(* IEC 61131-3 sources: Yaha/Documentation/Infomaterial/OSCAT/pcworx_basic_333/module_export (part 4) *)

(* ---- FT_PIDW.ST ---- *)
(*@PROPERTIES_EX@
TYPE: POU
LOCALE: 0
IEC_LANGUAGE: ST
PLC_TYPE: independent
PROC_TYPE: independent
GROUP: ENGINEERING.CONTROL
*)
(*@KEY@:DESCRIPTION*)
version 1.2	11. mar. 2009
programmer 	hugo
tested by	oscat

FT_PIDW is a PID controller with dynamic wind_up reset.
The PID controller works according to the fomula Y = KP *(IN + KI * INTEG(e) + DERIV(e) ).
a rst will reset the integrator to 0
lim_h and Lim_l set the possible output range of the internal integrator.
the output flags lim will signal that the output limits are active.

default values for KP = 1, KI = 1, ILIM_L = -1E37, iLIM_H = +1E38.
(*@KEY@:END_DESCRIPTION*)
FUNCTION_BLOCK FT_PIDW

(*Group:Default*)

VAR_INPUT
	IN :	REAL;
	KP :	REAL := 1.0;
	TN :	REAL := 1.0;
	TV :	REAL := 1.0;
	LIM_L :	REAL := -1.0E38;
	LIM_H :	REAL := 1.0E38;
	RST :	BOOL := FALSE;
END_VAR

VAR_OUTPUT
	Y :	REAL;
	LIM :	BOOL;
END_VAR

VAR
	integ :	INTEGRATE;
	diff :	FT_DERIV;
	YI :	REAL;
END_VAR

(*@KEY@: WORKSHEET
NAME: FT_PIDW
IEC_LANGUAGE: ST
*)
(* run the integrator *)
IF tn = 0.0 OR rst THEN
	integ(E := FALSE, Y := YI);
	YI := integ.Y;
	YI := 0.0;
ELSE
	integ(X := IN, K := 1.0 / TN, E := NOT LIM, Y := YI);
	YI := integ.Y;
END_IF;

(* add up integrator and linear part *)
Y := KP * (IN + YI);

(* run differentiator *)
diff(IN := IN, K := TV);

(* set lim before differentiator is added to stop integrator if necessary *)
IF Y > LIM_L AND Y < LIM_H THEN
	LIM := FALSE;
ELSE
	LIM := TRUE;
END_IF;

(* add differential part and limit output Y *)

Y := LIMIT(LIM_L, Y + KP * diff.out, LIM_H);

(* revision history
hm 3. jun. 2008 	rev 1.0
	original version

hm	5. nov. 2008	rev 1.1
	changed code to use integrate

hm	11. mar. 2009	rev 1.2
	real constants updated to new systax using dot

*)
(*@KEY@: END_WORKSHEET *)
END_FUNCTION_BLOCK

(* ---- FT_PIDWL.ST ---- *)
(*@PROPERTIES_EX@
TYPE: POU
LOCALE: 0
IEC_LANGUAGE: ST
PLC_TYPE: independent
PROC_TYPE: independent
GROUP: ENGINEERING.CONTROL
*)
(*@KEY@:DESCRIPTION*)
version 1.3	13. nov. 2009
programmer 	hugo
tested by	tobias

FT_PIDWL is a PID controller with dynamic wind_up reset.
The PID controller works according to the fomula Y = KP *(IN + KI * INTEG(e) + DERIV(e) ).
a rst will reset the integrator to 0
lim_h and Lim_l set the possible output range of the internal integrator.
the output flags lim will signal that the output limits are active.

default values for KP = 1, KI = 1, ILIM_L = -1E37, iLIM_H = +1E38.
(*@KEY@:END_DESCRIPTION*)
FUNCTION_BLOCK FT_PIDWL

(*Group:Default*)

VAR_INPUT
	IN :	REAL;
	KP :	REAL := 1.0;
	TN :	REAL := 1.0;
	TV :	REAL := 1.0;
	LIM_L :	REAL := -1.0E38;
	LIM_H :	REAL := 1.0E38;
	RST :	BOOL;
END_VAR

VAR_OUTPUT
	Y :	REAL;
	LIM :	BOOL;
END_VAR

VAR
	piwl :	FT_PIWL;
	diff :	FT_DERIV;
END_VAR

(*@KEY@: WORKSHEET
NAME: FT_PIDWL
IEC_LANGUAGE: ST
*)
(* if rst then *)
IF rst THEN
	piwl(rst := TRUE);
	piwl.RST := FALSE;
ELSE
	(* run PIWL controller first *)
	(* we need to check if TN = 0 and do alternative calls *)
	IF TN = 0.0 THEN
		piwl(in := IN * KP, KP := 1.0, KI := 0.0, LIM_L := LIM_L, LIM_H := LIM_H);
	ELSE
		piwl(in := IN * KP, KP := 1.0, KI := 1.0 / TN, LIM_L := LIM_L, LIM_H := LIM_H);
	END_IF;

	(* run differentiator and add_to_output *)
	diff(IN := IN, K := KP * TV);
	Y := piwl.Y + diff.out;

	(* limit the output *)
	IF Y < LIM_L THEN
		LIM := TRUE;
		Y := LIM_L;
	ELSIF Y > LIM_H THEN
		LIM := TRUE;
		Y := LIM_H;
	ELSE
		LIM := FALSE;
	END_IF;
END_IF;

(* revision history
hm 13. jun. 2008 	rev 1.0
	original version

hm	25. jan 2008	rev 1.1
	multiply differential part with KP

hm	11. mar. 2009	rev 1.2
	real constants updated to new systax using dot

hm	13. nov. 2009	rev 1.3
	fixed code for negative KP

*)
(*@KEY@: END_WORKSHEET *)
END_FUNCTION_BLOCK

(* ---- FT_PIW.ST ---- *)
(*@PROPERTIES_EX@
TYPE: POU
LOCALE: 0
IEC_LANGUAGE: ST
PLC_TYPE: independent
PROC_TYPE: independent
GROUP: ENGINEERING.CONTROL
*)
(*@KEY@:DESCRIPTION*)
version 1.0	3. jun 2008
programmer 	hugo
tested by	tobias

FT_PI is a PI controller.
The PID controller works according to the fomula Y = IN *(KP+ KI * INTEG(e) ).
a rst will reset the integrator to 0
ilim_h and iLim_l set the possible output range of the internal integrator.
the output flags lim will signal that the output limits are active.

default values for KP = 1, KI = 1, ILIM_L = -1E37, iLIM_H = +1E38.
(*@KEY@:END_DESCRIPTION*)
FUNCTION_BLOCK FT_PIW

(*Group:Default*)

VAR_INPUT
	IN :	REAL;
	KP :	REAL := 1.0;
	KI :	REAL := 1.0;
	LIM_L :	REAL := -1.0E38;
	LIM_H :	REAL := 1.0E38;
	RST :	BOOL := FALSE;
END_VAR

VAR_OUTPUT
	Y :	REAL;
	LIM :	BOOL;
END_VAR

VAR
	integ :	FT_INT;
END_VAR

(*@KEY@: WORKSHEET
NAME: FT_PIW
IEC_LANGUAGE: ST
*)
(* run integrator *)
integ(IN := IN, K := KI, RUN := NOT LIM, RST := RST);

(* set output value *)
Y := KP * IN + integ.Out;

(* check for limits *)
IF Y < LIM_L THEN
	Y := LIM_L;
	LIM := TRUE;
ELSIF Y > LIM_H THEN
	Y := LIM_H;
	LIM := TRUE;
ELSE
	LIM := FALSE;
END_IF;

(* revision history
hm 	3. jun. 2008 	rev 1.0
	original version

*)
(*@KEY@: END_WORKSHEET *)
END_FUNCTION_BLOCK

(* ---- FT_PIWL.ST ---- *)
(*@PROPERTIES_EX@
TYPE: POU
LOCALE: 0
IEC_LANGUAGE: ST
PLC_TYPE: independent
PROC_TYPE: independent
GROUP: ENGINEERING.CONTROL
*)
(*@KEY@:DESCRIPTION*)
version 1.3	11. mar. 2009
programmer 	hugo
tested by	oscat

FT_PIWL is a PI controller.
The PID controller works according to the fomula Y = IN *(KP+ KI * INTEG(e) ).
a rst will reset the integrator to 0
lim_h and Lim_l set the possible output range of the controller.
the output flag lim will signal that the output limits are active.
the integrator ist equipped with anti wind-up circuitry which limits trhe total output ranke to lim_l and lim_h

default values for KP = 1, KI = 1, ILIM_L = -1E37, iLIM_H = +1E38.

(*@KEY@:END_DESCRIPTION*)
FUNCTION_BLOCK FT_PIWL

(*Group:Default*)

VAR_INPUT
	IN :	REAL;
	KP :	REAL := 1.0;
	KI :	REAL := 1.0;
	LIM_L :	REAL := -1.0E38;
	LIM_H :	REAL := 1.0E38;
	RST :	BOOL;
END_VAR

VAR_OUTPUT
	Y :	REAL;
	LIM :	BOOL;
END_VAR

VAR
	init :	BOOL;
	tx :	UDINT;
	tc :	REAL;
	t_last :	UDINT;
	in_last :	REAL;
	i :	REAL;
	p :	REAL;
	T_PLC_US :	T_PLC_US;
END_VAR

(*@KEY@: WORKSHEET
NAME: FT_PIWL
IEC_LANGUAGE: ST
*)
(* initialize at power_up *)
IF NOT init OR RST THEN
	init := TRUE;
	in_last := in;
	T_PLC_US();
	t_last := T_PLC_US.T_PLC_US;
	i := 0.0;
	tc := 0.0;
ELSE
	(* read last cycle time in Microseconds *)
	T_PLC_US();
	tx := T_PLC_US.T_PLC_US;
	tc := UDINT_TO_REAL(tx - t_last);
	t_last := tx;

	(* calculate proportional part *)
	p := KP * IN;

	(* run integrator *)
	i := (IN + in_last) * 5.0E-7 * KI * tc + i;
	in_last := IN;

	(* calculate output Y *)
	Y := p + i;

	(* check output for limits *)
	IF Y >= LIM_H THEN
		Y := LIM_H;
		IF ki <> 0.0 THEN
			i := LIM_H - p;
		ELSE
			i := 0.0;
		END_IF;
		LIM := TRUE;
	ELSIF Y <= LIM_L THEN
		Y := LIM_L;
		IF ki <> 0.0 THEN
			i := LIM_L - p;
		ELSE
			i := 0.0;
		END_IF;
		LIM := TRUE;
	ELSE
		LIM := FALSE;
	END_IF;
END_IF;

(* revision history
hm 13. jun. 2008 	rev 1.0
	original version

hm	27. oct. 2008	rev 1.1
	integrator will not be adjusted when ki = 0

hm	25. jan 2009	rev 1.2
	module will also work with negative K

hm	11. mar. 2009	rev 1.3
	real constants updated to new systax using dot

*)
(*@KEY@: END_WORKSHEET *)
END_FUNCTION_BLOCK

(* ---- FT_PROFILE.ST ---- *)
(*@PROPERTIES_EX@
TYPE: POU
LOCALE: 0
IEC_LANGUAGE: ST
PLC_TYPE: independent
PROC_TYPE: independent
GROUP: ENGINEERING.AUTOMATION
*)
(*@KEY@:DESCRIPTION*)
version 1.1	15 sep 2007
programmer 	tobias
tested by	hugo

FT_Profile generates an output signal which is defined by values over a time scale.
the different values are connected by ramps between the individual values.
a rising edge on E starts the output signal generation and E = True can delay time_3 / value_3 as long as it stays true.
an additional multiplier K can be used to multiply the output and an offset O can be added to the output dynamically.
(*@KEY@:END_DESCRIPTION*)
FUNCTION_BLOCK FT_PROFILE

(*Group:Default*)

VAR_INPUT
	K :	REAL := 1.0;
	O :	REAL := 0.0;
	M :	REAL := 1.0;
	E :	BOOL;
	VALUE_0 :	REAL;
	TIME_1 :	TIME;
	VALUE_1 :	REAL;
	TIME_2 :	TIME;
	VALUE_2 :	REAL;
	TIME_3 :	TIME;
	VALUE_3 :	REAL;
	TIME_10 :	TIME;
	VALUE_10 :	REAL;
	TIME_11 :	TIME;
	VALUE_11 :	REAL;
	TIME_12 :	TIME;
	VALUE_12 :	REAL;
	TIME_13 :	TIME;
	VALUE_13 :	REAL;
END_VAR

VAR_OUTPUT
	Y :	REAL;
	RUN :	BOOL;
	ET :	TIME;
END_VAR

VAR
	tx :	TIME;
	edge :	BOOL;
	state :	INT;
	ta :	TIME;
	tb :	TIME;
	t0 :	TIME;
	temp :	REAL;
	va :	REAL;
	vb :	REAL;
	T_PLC_MS :	T_PLC_MS;
END_VAR

(*@KEY@: WORKSHEET
NAME: FT_PROFILE
IEC_LANGUAGE: ST
*)
(* read system time *)
T_PLC_MS();
tx:= UDINT_TO_TIME(T_PLC_MS.T_PLC_MS);

(* determine start condition *)
IF E AND NOT edge THEN
	RUN := TRUE;
	ET := t#0s;
	t0 := tx;
	ta := tx;
	tb := multime(time_1, M);
	va := value_0;
	vb := value_1;
	temp := value_0;
	state := 1;
END_IF;
edge := E;

(* generate startup profile *)
IF run THEN
	CASE state OF
		1:	IF tx - ta >= tb THEN
				ta := ta + tb;
				tb := multime(time_2 - time_1, M);
				va := value_1;
				vb := value_2;
				temp := value_1;
				state := 2;
			ELSE
				temp := ((vb - va) * TIME_TO_REAL(tx - ta) / TIME_TO_REAL(tb) + va);
			END_IF;
		2:	IF tx - ta >= tb THEN
				ta := ta + tb;
				tb := multime(time_3 - time_2, M);
				va := value_2;
				vb := value_3;
				temp := value_2;
				state := 3;
			ELSE
				temp := ((vb - va) * TIME_TO_REAL(tx - ta) / TIME_TO_REAL(tb) + va);
			END_IF;
		3:	IF tx - ta >= tb THEN
				ta := ta + tb;
				tb := multime(time_10 - time_3, M);
				va := value_3;
				vb := value_10;
				temp := value_3;
				state := 4;
			ELSE
				temp := ((vb - va) * TIME_TO_REAL(tx - ta) / TIME_TO_REAL(tb) + va);
			END_IF;
		4 :	IF tx - ta >= tb THEN
				ta := ta + tb;
				tb := multime(time_11 - time_10, M);
				va := value_10;
				vb := value_11;
				temp := value_10;
				IF E THEN state := 5; ELSE state := 6; END_IF;
			ELSE
				temp := ((vb - va) * TIME_TO_REAL(tx - ta) / TIME_TO_REAL(tb) + va);
			END_IF;
		5:	(* extend the signal while E is true *)
			IF E THEN
				ta := tx;
			ELSE
				state := 6;
			END_IF;
		6:	IF tx - ta >= tb THEN
				ta := ta + tb;
				tb := multime(time_12 - time_11, M);
				va := value_11;
				vb := value_12;
				temp := value_11;
				state := 7;
			ELSE
				temp := ((vb - va) * TIME_TO_REAL(tx - ta) / TIME_TO_REAL(tb) + va);
			END_IF;
		7:	IF tx - ta >= tb THEN
				ta := ta + tb;
				tb := multime(time_13 - time_12, M);
				va := value_12;
				vb := value_13;
				temp := value_12;
				state := 8;
			ELSE
				temp := ((vb - va) * TIME_TO_REAL(tx - ta) / TIME_TO_REAL(tb) + va);
			END_IF;
		8:	IF tx - ta >= tb THEN
				temp := value_13;
				run := FALSE;
			ELSE
				temp := ((vb - va) * TIME_TO_REAL(tx - ta) / TIME_TO_REAL(tb) + va);
			END_IF;
	END_CASE;
	Y := temp * K + O;
	ET := tx - t0;
END_IF;

(* revision history
hm	27 feb 2007		rev 1.0
	original version

hm	15. sep2007		rev 1.1
	replaced Time() with T_PLC_MS for compatibility and performance reasons

*)
(*@KEY@: END_WORKSHEET *)
END_FUNCTION_BLOCK

(* ---- FT_PT1.ST ---- *)
(*@PROPERTIES_EX@
TYPE: POU
LOCALE: 0
IEC_LANGUAGE: ST
PLC_TYPE: independent
PROC_TYPE: independent
GROUP: ENGINEERING.CONTROL
*)
(*@KEY@:DESCRIPTION*)
version 1.11	18. jan. 2011
programmer 		hugo
tested by		oscat

FT_PT1 is an low pass filter with a programmable time T and faktor K.

(*@KEY@:END_DESCRIPTION*)
FUNCTION_BLOCK FT_PT1

(*Group:Default*)

VAR_INPUT
	IN :	REAL;
	T :	TIME;
	K :	REAL := 1.0;
END_VAR

VAR_OUTPUT
	OUT :	REAL;
END_VAR

VAR
	last :	UDINT;
	tx :	UDINT;
	init :	BOOL;
	T_PLC_US :	T_PLC_US;
END_VAR

(*@KEY@: WORKSHEET
NAME: FT_PT1
IEC_LANGUAGE: ST
*)
(* read system time *)
T_PLC_US();
tx:= T_PLC_US.T_PLC_US;

(* startup initialisation *)
IF NOT init OR T = t#0s THEN
	init := TRUE;
	out := K * in;
ELSE
	out := out + (in * K - out) * UDINT_TO_REAL(Tx - last) / TIME_TO_REAL(T) * 1.0E-3;
	IF ABS(out) < 1.0E-20 THEN out := 0.0; END_IF;
END_IF;
last := tx;

(*
hm 1.1.2007	rev 1.1
	corrected error while startup value was not correct
	for very small time values real output would run out of range.

hm 3.1.2007	rev 1.2
	corrected an error for falling edge failures.
	added output faktor K.

hm 27. 2. 2007	rev 1.3
	output will be input during init for definitive startup condition.

hm	15.9.2007	rev 1.4
	changed time() to T_PLC_US() for compatibilitxy resons
	increased internal accuracy to Microseconds instead of Milliseconds

hm	23. oct 2007	rev 1.5
	added out := in to the init statements

hm	30. nov 2007	rev 1.6
	changed out to be K * in during initialization

hm	5. jan 2008	rev 1.7
	improved code for better performance

hm	16. mar. 2008	rev 1.8
	added type conversion to avoid warning under codesys 3.0

hm	14. jun. 2008	rev 1.9
	improved code

hm	11. mar. 2009	rev 1.10
	real constants updated to new systax using dot

hm	18. jan. 2011	rev 1.11
	avoid underrun of out
*)
(*@KEY@: END_WORKSHEET *)
END_FUNCTION_BLOCK

(* ---- FT_PT2.ST ---- *)
(*@PROPERTIES_EX@
TYPE: POU
LOCALE: 0
IEC_LANGUAGE: ST
PLC_TYPE: independent
PROC_TYPE: independent
GROUP: ENGINEERING.CONTROL
*)
(*@KEY@:DESCRIPTION*)
version 1.5	11. mar. 2009
programmer 	hugo
tested by	oscat

FT_PT2 is a 2nd grade filter with programmable times T, D and faktor K.
(*@KEY@:END_DESCRIPTION*)
FUNCTION_BLOCK FT_PT2

(*Group:Default*)

VAR_INPUT
	IN :	REAL;
	T :	TIME;
	D :	REAL;
	K :	REAL := 1.0;
END_VAR

VAR_OUTPUT
	OUT :	REAL;
END_VAR

VAR
	init :	BOOL;
	int1 :	INTEGRATE;
	int2 :	INTEGRATE;
	tn :	REAL;
	I1 :	REAL;
	I2 :	REAL;
	tn2 :	REAL;
END_VAR

(*@KEY@: WORKSHEET
NAME: FT_PT2
IEC_LANGUAGE: ST
*)
(* startup initialisation *)
IF NOT init OR T = T#0s THEN
	init := TRUE;
	out := K * in;
	I2 := out;
ELSE
	TN := TIME_TO_REAL(T) / 1000.0;
	tn2 := TN * TN;
	int1(X := in * K / tn2 - I1 * 0.5 * D / TN - I2 / TN2, Y := I1);
	I1 := int1.Y;
	int2(X := I1,Y := I2);
	I2 := int2.Y;
	out := I2;
END_IF;

(* revision history

15.1.2007 hm		rev 1.1
	changed formula to new more acurate formula

hm 15.9.2007		rev 1.2
	deleted unused code for init system time reading tx

hm	30.11.2007	rev 1.3
	changed out to be K * in during initialization
	avoind divide by 0 if tn = 0

hm	3. nov. 2008	rev 1.4
	optimized code and fixed a problem with init

hm	11. mar. 2009	rev 1.5
	real constants updated to new systax using dot

*)
(*@KEY@: END_WORKSHEET *)
END_FUNCTION_BLOCK

(* ---- FT_RMP.ST ---- *)
(*@PROPERTIES_EX@
TYPE: POU
LOCALE: 0
IEC_LANGUAGE: ST
PLC_TYPE: independent
PROC_TYPE: independent
GROUP: MATHEMATICAL.FUNCTIONS
*)
(*@KEY@:DESCRIPTION*)
version 1.4	25 jan 2008
programmer 	oscat
tested BY	oscat

this ramp function follows an input signal with a linear ramp up or down, the up or down speed can be set with KF and KR.
a K factor of 1 means 1 unit per second on the output. K factors can only be positive and not negative.
a busy output signals the ramp is running or busy false means the in value is present on the output.
a rmp input false means the output follows the input dierctly while a rmp = true means the output follows the input with a ramp.
a updn output signal the directon of the ramp (up or down).
(*@KEY@:END_DESCRIPTION*)
FUNCTION_BLOCK FT_RMP

(*Group:Default*)

VAR_INPUT
	RMP :	BOOL := TRUE;
	IN :	REAL;
	KR :	REAL;
	KF :	REAL;
END_VAR

VAR_OUTPUT
	OUT :	REAL;
	BUSY :	BOOL;
	UD :	BOOL;
END_VAR

VAR
	tx :	TIME;
	last :	TIME;
	init :	BOOL;
	T_PLC_MS :	T_PLC_MS;
END_VAR

(*@KEY@: WORKSHEET
NAME: FT_RMP
IEC_LANGUAGE: ST
*)
(* read system time *)
T_PLC_MS();
tx:= UDINT_TO_TIME(T_PLC_MS.T_PLC_MS) - last;

IF NOT init THEN
	init := TRUE;
	last := tx;
	tx := t#0s;
	out := in;
END_IF;
IF NOT rmp THEN
	out := in;
	busy := FALSE;
ELSIF out > in THEN
	(* ramp down *)
	out := out - TIME_TO_REAL(tx) * 0.001 * KF;
	out := MAX(in, out);
ELSIF out < in THEN
	(* ramp up *)
	out := out + TIME_TO_REAL(tx) * 0.001 * KR;
	out := MIN(in, out);
END_IF;

(* set busy and dir flags *)
IF out < in THEN
	busy := TRUE;
	ud := TRUE;
ELSIF out > in THEN
	busy := TRUE;
	ud := FALSE;
ELSE
	busy := FALSE;
END_IF;
last := last + tx;

(* revision history:

hm 8.10.2006			rev 1.1
	added ud output

hm 12. feb 2007		rev 1.2
	added init variable and corrected a possible startup problem

hm	17. sep 2007	rev 1.3
	replaced time() with t_plc_ms() for compatibility reasons

hm	25. jan 2008	rev 1.4
	performance improvements
	allow KR and KF to be 0
*)
(*@KEY@: END_WORKSHEET *)
END_FUNCTION_BLOCK

(* ---- FT_TN16.ST ---- *)
(*@PROPERTIES_EX@
TYPE: POU
LOCALE: 0
IEC_LANGUAGE: ST
PLC_TYPE: independent
PROC_TYPE: independent
GROUP: ENGINEERING.CONTROL
*)
(*@KEY@:DESCRIPTION*)
version 1.1	16 sep 2007
programmer 	hugo
tested by	tobias

FT_TN16 is delay function, it will delay a signal by a specified time : T and will store 16 values of in before they are put thru to out.
for higher or lower resolution please use FT_TN8 or FT_TN64 instead.
(*@KEY@:END_DESCRIPTION*)
FUNCTION_BLOCK FT_TN16

(*Group:Default*)

VAR_INPUT
	IN :	REAL;
	T :	TIME;
END_VAR

VAR_OUTPUT
	OUT :	REAL;
	TRIG :	BOOL;
END_VAR

VAR
	length :	INT := 16;
	X :	oscat_arr_0_15;
	cnt :	INT;
	last :	TIME;
	tx :	TIME;
	init :	BOOL;
	T_PLC_MS :	T_PLC_MS;
END_VAR

(*@KEY@: WORKSHEET
NAME: FT_TN16
IEC_LANGUAGE: ST
*)
(* read system time *)
T_PLC_MS();
tx:= UDINT_TO_TIME(T_PLC_MS.T_PLC_MS);

trig := FALSE;
IF NOT init THEN
	x[cnt] := in;
	init := TRUE;
	last := tx;
ELSIF tx - last >= T / INT_TO_TIME(length) THEN
	IF cnt = length - 1 THEN cnt := 0; ELSE cnt := cnt + 1; END_IF;
	Out := X[cnt];
	x[cnt] := in;
	last := tx;
	Trig := TRUE;
END_IF;

(* revision history
hm		1. jan 2007		rev 1.0
	original version

hm		16. sep 2007	rev 1.1
	changes time() to T_plc_ms() for compatibility reasons

*)
(*@KEY@: END_WORKSHEET *)
END_FUNCTION_BLOCK

(* ---- FT_TN64.ST ---- *)
(*@PROPERTIES_EX@
TYPE: POU
LOCALE: 0
IEC_LANGUAGE: ST
PLC_TYPE: independent
PROC_TYPE: independent
GROUP: ENGINEERING.CONTROL
*)
(*@KEY@:DESCRIPTION*)
version 1.1	15 sep 2007
programmer 	hugo
tested by	tobias

FT_TN7 is delay function, it will delay a signal by a specified time : T and will store 64 values of in before they are put thru to out.
if lower resolution is needed, pls use FT_TN8 or FT_TN16 instead.
(*@KEY@:END_DESCRIPTION*)
FUNCTION_BLOCK FT_TN64

(*Group:Default*)

VAR_INPUT
	IN :	REAL;
	T :	TIME;
END_VAR

VAR_OUTPUT
	OUT :	REAL;
	TRIG :	BOOL;
END_VAR

VAR
	length :	INT := 64;
	X :	oscat_FT_TN64_array;
	cnt :	INT;
	last :	TIME;
	tx :	TIME;
	init :	BOOL;
	T_PLC_MS :	T_PLC_MS;
END_VAR

(*@KEY@: WORKSHEET
NAME: FT_TN64
IEC_LANGUAGE: ST
*)
(* read system time *)
T_PLC_MS();
tx:= UDINT_TO_TIME(T_PLC_MS.T_PLC_MS);

trig := FALSE;
IF NOT init THEN
	x[cnt] := in;
	init := TRUE;
	last := tx;
ELSIF tx - last >= T / INT_TO_TIME(length) THEN
	IF cnt = length - 1 THEN cnt := 0; ELSE cnt := cnt + 1; END_IF;
	Out := X[cnt];
	x[cnt] := in;
	last := tx;
	trig := TRUE;
END_IF;

(* revision history
hm		1. jan 2007		rev 1.0
	original version

hm		16. sep 2007	rev 1.1
	changes time() to T_plc_ms() for compatibility reasons

*)
(*@KEY@: END_WORKSHEET *)
END_FUNCTION_BLOCK

(* ---- FT_TN8.ST ---- *)
(*@PROPERTIES_EX@
TYPE: POU
LOCALE: 0
IEC_LANGUAGE: ST
PLC_TYPE: independent
PROC_TYPE: independent
GROUP: ENGINEERING.CONTROL
*)
(*@KEY@:DESCRIPTION*)
version 1.1	15 Sep 2007
programmer 	hugo
tested by	tobias

FT_TN8 is delay function, it will delay a signal by a specified time : T and will store 8 values of in before they are put thru to out.
if higher resolution is needed, pls use FT_TN16 or FT_TN64 instead.
(*@KEY@:END_DESCRIPTION*)
FUNCTION_BLOCK FT_TN8

(*Group:Default*)

VAR_INPUT
	IN :	REAL;
	T :	TIME;
END_VAR

VAR_OUTPUT
	OUT :	REAL;
	TRIG :	BOOL;
END_VAR

VAR
	length :	INT := 8;
	X :	oscat_arr_0_7;
	cnt :	INT;
	last :	TIME;
	tx :	TIME;
	init :	BOOL;
	T_PLC_MS :	T_PLC_MS;
END_VAR

(*@KEY@: WORKSHEET
NAME: FT_TN8
IEC_LANGUAGE: ST
*)
T_PLC_MS();
tx:= UDINT_TO_TIME(T_PLC_MS.T_PLC_MS);

trig := FALSE;
IF NOT init THEN
	x[cnt] := in;
	init := TRUE;
	last := tx;
ELSIF tx - last >= T / INT_TO_TIME(length) THEN
	IF cnt = length - 1 THEN cnt := 0; ELSE cnt := cnt + 1; END_IF;
	Out := X[cnt];
	x[cnt] := in;
	last := tx;
	trig := TRUE;
END_IF;

(* revision history
hm		1. jan 2007		rev 1.0
	original version

hm		16. sep 2007	rev 1.1
	changes time() to T_plc_ms() for compatibility reasons

*)
(*@KEY@: END_WORKSHEET *)
END_FUNCTION_BLOCK

(* ---- GEN_BIT.ST ---- *)
(*@PROPERTIES_EX@
TYPE: POU
LOCALE: 0
IEC_LANGUAGE: ST
PLC_TYPE: independent
PROC_TYPE: independent
GROUP: LOGIC.GENERATORS
*)
(*@KEY@:DESCRIPTION*)
version 1.2	14. mar. 2009
programmer 	hugo
tested by	tobias

gen_bit is 4 bit sequencial pattern generator with 4 DWORD inputs and 4 serial outputs.
with the first clock pulse after a reset or after power on, bit 0 of the input DWORDS IN is present on the Outputs Q and the next clock cycle shifts to Bit 1 and so on.
the input steps defines how many bits of the input dwords will be shifted to the outputs. the sequence can be repetive when rep = 0 or any amount of repetitions can be defined with input rep.

(*@KEY@:END_DESCRIPTION*)
FUNCTION_BLOCK GEN_BIT

(*Group:Default*)

VAR_INPUT
	IN0 :	DWORD;
	IN1 :	DWORD;
	IN2 :	DWORD;
	IN3 :	DWORD;
	CLK :	BOOL;
	STEPS :	INT;
	REP :	INT;
	RST :	BOOL;
END_VAR

VAR_OUTPUT
	Q0 :	BOOL;
	Q1 :	BOOL;
	Q2 :	BOOL;
	Q3 :	BOOL;
	CNT :	INT;
	RUN :	BOOL;
END_VAR

VAR
	r0 :	DWORD;
	r1 :	DWORD;
	r2 :	DWORD;
	r3 :	DWORD;
	rx :	INT := 1;
END_VAR

(*@KEY@: WORKSHEET
NAME: GEN_BIT
IEC_LANGUAGE: ST
*)
(* check if number of runs is finished or rep = 0 which means continuous *)

IF clk AND NOT rst THEN
	run := (rep = 0) OR (rx <= rep);
	IF run THEN
		(* check for step counter reached and reset to 0 if cnt = steps *)
		IF cnt = steps THEN
			cnt := 0;
		END_IF;

		(* when cnt = 0 then reload the inputs into the registers *)
		IF cnt = 0 THEN
			r0 := in0;
			r1 := in1;
			r2 := in2;
			r3 := in3;
		END_IF;

		(* when cnt < steps, shift the lowest bits to the outputs *)
		IF (cnt < steps) THEN
            Q0 := BIT_OF_DWORD(r0,0); (* Q0 := r0.X0; *)
            Q1 := BIT_OF_DWORD(r1,0); (* Q1 := r1.X0; *)
            Q2 := BIT_OF_DWORD(r2,0); (* Q2 := r2.X0; *)
            Q3 := BIT_OF_DWORD(r3,0); (* Q3 := r3.X0; *)
			r0 := SHR(r0,1);
			r1 := SHR(r1,1);
			r2 := SHR(r2,1);
			r3 := SHR(r3,1);
		END_IF;

		(* increment the step counter *)
		cnt := cnt +1;
		IF (cnt = steps) AND (rep <> 0) THEN rx := rx +1; END_IF;
		IF (rx > rep) AND (rep <> 0) THEN run := FALSE; END_IF;
	END_IF;
ELSE
	IF rst THEN
		run := FALSE;
		Q0 := FALSE;
		Q1 := FALSE;
		Q2 := FALSE;
		Q3 := FALSE;
		r0 := DWORD#0;
		r1 := DWORD#0;
		r2 := DWORD#0;
		r3 := DWORD#0;
		cnt := 0;
		rx := 1;
	END_IF;
END_IF;

(* revision histroy
hm	4 aug 2006	rev 1.0
	original version

hm 15. oct. 2008	rev 1.1
	improved performance

hm	14. mar. 2009	rev 1.2
	removed double assignments

*)

(*@KEY@: END_WORKSHEET *)
END_FUNCTION_BLOCK

(* ---- GEN_PULSE.ST ---- *)
(*@PROPERTIES_EX@
TYPE: POU
LOCALE: 0
IEC_LANGUAGE: ST
PLC_TYPE: independent
PROC_TYPE: independent
GROUP: ENGINEERING.SIGNAL_GENERATORS
*)
(*@KEY@:DESCRIPTION*)
version 1.5	8. apr. 2011
programmer 	hugo
tested by	oscat

GEN_PULSE uses the internal sps timer to generate a continuous output waveform with programmable high and low time.
the accuracy of gen_pulse is depending on the system timer.
when time is 0 the high and low times are exactly one cycle.
ENQ = TRUE will start and ENQ = FALSE will stop the generator.
(*@KEY@:END_DESCRIPTION*)
FUNCTION_BLOCK GEN_PULSE

(*Group:Default*)

VAR_INPUT
	ENQ :	BOOL := TRUE;
	PTH :	TIME;
	PTL :	TIME;
END_VAR

VAR_OUTPUT
	Q :	BOOL;
END_VAR

VAR
	T_PLC_MS :	T_PLC_MS;
	tx :	TIME;
	tn :	TIME;
	init :	BOOL;
END_VAR

(*@KEY@: WORKSHEET
NAME: GEN_PULSE
IEC_LANGUAGE: ST
*)
IF enq THEN
	T_PLC_MS();	(* read system timer *)
	tx:= UDINT_TO_TIME(T_PLC_MS.T_PLC_MS);
	IF NOT init THEN init := TRUE; tn := tx; END_IF;
	IF tx - tn >= SEL(Q, PTL, PTH) THEN
		tn := tn + SEL(Q, PTL, PTH);
		Q := NOT Q;
	END_IF;
ELSE
	Q := FALSE;
	init := FALSE;
END_IF;

(* revision history
hm	29. jun. 2008	rev 1.0
	original version

hm	23. nov. 2008	rev 1.1
	set default for enq to be true

hm	18. jul. 2009	rev 1.2
	improved performance

hm	13. nov. 2009	rev 1.3
	corrected error

hm	16. feb. 2011	rev 1.4
	corrected an error when timer overflows

hm	8. apr. 2011	rev 1.5
	ptl and pth was exchanged
*)
(*@KEY@: END_WORKSHEET *)
END_FUNCTION_BLOCK

(* ---- GEN_PW2.ST ---- *)
(*@PROPERTIES_EX@
TYPE: POU
LOCALE: 0
IEC_LANGUAGE: ST
PLC_TYPE: independent
PROC_TYPE: independent
GROUP: ENGINEERING.SIGNAL_GENERATORS
*)
(*@KEY@:DESCRIPTION*)
version 1.1	14. mar. 2009
programmer 	hugo
tested by	oscat

GEN_PW2 generates a time TH? followed by a time TL?.
the input ts selects between 2 sets of timings for the operation.

(*@KEY@:END_DESCRIPTION*)
FUNCTION_BLOCK GEN_PW2

(*Group:Default*)

VAR_INPUT
	ENQ :	BOOL;
	TH1 :	TIME;
	TL1 :	TIME;
	TH2 :	TIME;
	TL2 :	TIME;
	TS :	BOOL;
END_VAR

VAR_OUTPUT
	Q :	BOOL;
	TH :	TIME;
	TL :	TIME;
END_VAR

VAR
	T_PLC_MS :	T_PLC_MS;
	t_high :	TIME;
	t_low :	TIME;
	tx :	TIME;
	start :	TIME;
	init :	BOOL;
	et :	TIME;
END_VAR

(*@KEY@: WORKSHEET
NAME: GEN_PW2
IEC_LANGUAGE: ST
*)
(* read system time and prepare input data *)
T_PLC_MS();
tx:= UDINT_TO_TIME(T_PLC_MS.T_PLC_MS);

(* startup initialization *)
IF NOT init THEN
	start := tx;
	init := TRUE;
	TH := T#0s;
	TL := T#0s;
END_IF;

(* timing selection *)
IF TS THEN
	t_high := TH2;
	t_low := TL2;
ELSE
	t_high := TH1;
	t_low := TL1;
END_IF;

(* normal operation *)
IF ENQ THEN
	et := tx - start;
	IF NOT Q THEN
		IF et >= t_low THEN
			Q := TRUE;
			start := tx;
			TL := T#0s;
		ELSE
			TL := et;
		END_IF;
	ELSE
		IF et >= t_high THEN
			Q := FALSE;
			start := tx;
			TH := T#0s;
		ELSE
			TH := et;
		END_IF;
	END_IF;
ELSE
	Q := FALSE;
	TH := T#0s;
	TL := T#0s;
	start := tx;
END_IF;

(* revision history
hm	26. sep. 2008	rev 1.0
	original version

hm	14. mar. 2009	rev 1.1
	removed double assignments

*)
(*@KEY@: END_WORKSHEET *)
END_FUNCTION_BLOCK

(* ---- GEN_RDM.ST ---- *)
(*@PROPERTIES_EX@
TYPE: POU
LOCALE: 0
IEC_LANGUAGE: ST
PLC_TYPE: independent
PROC_TYPE: independent
GROUP: ENGINEERING.SIGNAL_GENERATORS
*)
(*@KEY@:DESCRIPTION*)
version 1.1	16 sep 2007
programmer 	oscat
tested BY	oscat

this signal generator generates a random output. The signal is defined by period time (PT),
amplitude (AM), offset (OS).
The Output waveform will have its max peak at AM/2 + OS and its minimum peak at -AM/2 + OS.
The period time PT defines how often the output signal will jump to a new randow value.
The Output Q will be true for one cycle anytime the output OUT has changed
(*@KEY@:END_DESCRIPTION*)
FUNCTION_BLOCK GEN_RDM

(*Group:Default*)

VAR_INPUT
	PT :	TIME;
	AM :	REAL := REAL#1.0;
	OS :	REAL;
END_VAR

VAR_OUTPUT
	Q :	BOOL;
	Out :	REAL;
END_VAR

VAR
	tx :	TIME;
	last :	TIME;
	init :	BOOL;
	T_PLC_MS :	T_PLC_MS;
	FB_rdm :	rdm;
END_VAR

(*@KEY@: WORKSHEET
NAME: GEN_RDM
IEC_LANGUAGE: ST
*)
(* read system time and prepare input data *)
T_PLC_MS();
tx:= UDINT_TO_TIME(T_PLC_MS.T_PLC_MS) - last;

(* init section *)
IF NOT init THEN
	init := TRUE;
	last := tx;
	tx := t#0s;
END_IF;

(* add last if one cycle is finished *)
IF tx >= pt THEN
	last := last + pt;
	tx := tx - pt;

	(* generate output signal *)
    FB_rdm(last:=0.0);
	out := am * (FB_rdm.RDM - 0.5) + os;
	q := TRUE;
ELSE
	q := FALSE;
END_IF;

(* revision history

hm	7.2.2007		rev 1.0
	original version

hm	16.9.2007		rev 1.1
	changes time() to T_plc_ms() for compatibility reasons

*)
(*@KEY@: END_WORKSHEET *)
END_FUNCTION_BLOCK

(* ---- GEN_RDT.ST ---- *)
(*@PROPERTIES_EX@
TYPE: POU
LOCALE: 0
IEC_LANGUAGE: ST
PLC_TYPE: independent
PROC_TYPE: independent
GROUP: ENGINEERING.SIGNAL_GENERATORS
*)
(*@KEY@:DESCRIPTION*)
version 1.1	16 mar. 2008
programmer 	J. Schohaus
tested by	Hugo

RDMT generates a defined pulse with pulse width TP_Q at random times. the random time will be defined with an minimum and maximum time.
(*@KEY@:END_DESCRIPTION*)
FUNCTION_BLOCK GEN_RDT

(*Group:Default*)

VAR_INPUT
	ENABLE :	BOOL := TRUE;
	MIN_TIME_MS :	TIME := t#1s;(*min Taktzeit*)
	MAX_TIME_MS :	TIME := t#1.2s;(*Max Taktzeit*)
	TP_Q :	TIME := t#100ms;(*Zeit Ausgang auf TRUE*)
END_VAR

VAR_OUTPUT
	XQ :	BOOL;
END_VAR

VAR
	tonRDMTimer :	TON;(*Zeitbaustein Taktgenerator*)
	tof_xQ :	TOF;(*Ausschaltverzögerung Taktgenerator*)
	tRDMTime :	TIME;(*Sollzeit*)
	rRDMTime :	REAL;(*Zufallswert Timer*)
	rdm_1 :	rdm;
END_VAR

(*@KEY@: WORKSHEET
NAME: GEN_RDT
IEC_LANGUAGE: ST
*)
tonRDMTimer(IN:=Enable,PT:=tRDMTime);
tof_xQ(IN := tonRDMTimer.Q,PT:=TP_Q);
XQ := tof_xq.Q;
IF tonRDMTimer.Q THEN
	xQ := TRUE ;
    rdm_1(last:=rRDMTime);
    rRDMTime:= rdm_1.RDM;

	tRDMTime := REAL_TO_TIME(rRDMTime * TIME_TO_REAL(Max_Time_ms - Min_Time_ms) + TIME_TO_REAL(Min_Time_ms));
	tonRDMTimer (IN:=FALSE);
END_IF;

(* revision history
J. Schohaus	19. nov 2007	rev 1.0
	origial version

hm	16. mar. 2008			rev 1.1
	added type conversion to avoid warnings under codesys 3.0
*)
(*@KEY@: END_WORKSHEET *)
END_FUNCTION_BLOCK

(* ---- GEN_RMP.ST ---- *)
(*@PROPERTIES_EX@
TYPE: POU
LOCALE: 0
IEC_LANGUAGE: ST
PLC_TYPE: independent
PROC_TYPE: independent
GROUP: ENGINEERING.SIGNAL_GENERATORS
*)
(*@KEY@:DESCRIPTION*)
version 1.4	10. mar. 2009
programmer 	oscat
tested BY	oscat

this signal generator generates a ramp wave output. The ramp wave signal is defined by period time (PT),
amplitude (AM), offset (OS) and a specific delay for the output signal (DL).
The Output waveform will have its minimum peak at OS and its maximum peak at AM + OS.
The delay input can delay a signal up to PT, this can be useful to synchronize different generators
and generate interleaving signals.
in addition to the analog output Out there is a second boolean output Q with is true for one cycle when the ramp starts.

(*@KEY@:END_DESCRIPTION*)
FUNCTION_BLOCK GEN_RMP

(*Group:Default*)

VAR_INPUT
	PT :	TIME := T#1s;
	AM :	REAL := REAL#1.0;
	OS :	REAL;
	DL :	REAL;
END_VAR

VAR_OUTPUT
	Q :	BOOL;
	OUT :	REAL;
END_VAR

VAR
	tx :	TIME;
	last :	TIME;
	init :	BOOL;
	temp :	REAL;
	ltemp :	REAL;
	T_PLC_MS :	T_PLC_MS;
END_VAR

(*@KEY@: WORKSHEET
NAME: GEN_RMP
IEC_LANGUAGE: ST
*)
(* read system time and prepare input data *)
T_PLC_MS();
tx:= UDINT_TO_TIME(T_PLC_MS.T_PLC_MS) - last;
DL := modR(dl,1.0);
IF dl < 0.0 THEN dl := 1.0 - dl; END_IF;

(* init section *)
IF NOT init THEN
	init := TRUE;
	last := tx;
	tx := t#0s;
END_IF;

(* add last if one cycle is finished *)
IF tx >= pt THEN
	last := last + pt;
	tx := tx - pt;
END_IF;

(* generate sine wave *)
ltemp := temp;
IF pt > t#0s THEN temp := fract(TIME_TO_REAL(tx + multime(pt, dl)) / TIME_TO_REAL(pt)); END_IF;
out := am * temp + os;

(* boolean output Q *)
Q := temp < ltemp;

(* revision history
hm	3. mar 2007		rev 1.0
	original version

hm	17 sep 2007		rev 1.1
	replaced time() with t_plc_ms for compatibilitx reasons

hm	27. nov 2007	rev 1.2
	avoid divide by 0 when pt = 0

ks	26. oct. 2008	rev 1.3
	code optimization

hm	10. mar. 2009	rev 1.4
	changed real constants to use dot syntax
*)
(*@KEY@: END_WORKSHEET *)
END_FUNCTION_BLOCK

(* ---- GEN_SIN.ST ---- *)
(*@PROPERTIES_EX@
TYPE: POU
LOCALE: 0
IEC_LANGUAGE: ST
PLC_TYPE: independent
PROC_TYPE: independent
GROUP: ENGINEERING.SIGNAL_GENERATORS
*)
(*@KEY@:DESCRIPTION*)
version 1.6	11. mar. 2009
programmer 	oscat
tested BY	oscat

this signal generator generates a sine wave output. The sine wave signal is defined by period time (PT),
amplitude (AM), offset (OS) and a specific delay for the output signal (DL).
The Output waveform will have its max peak at AM/2 + OS and its minimum peak at -AM/2 + OS.
The delay input can delay a signal up to PT, this can be useful to synchronize different generators
and generate interleaving signals. A Cos wave can be generated accordingly.
in addition to a analog output Out there is a second boolean output Q with the corresponding binary signal.

(*@KEY@:END_DESCRIPTION*)
FUNCTION_BLOCK GEN_SIN

(*Group:Default*)

VAR_INPUT
	PT :	TIME;
	AM :	REAL := REAL#1.0;
	OS :	REAL;
	DL :	REAL;
END_VAR

VAR_OUTPUT
	Q :	BOOL;
	Out :	REAL;
END_VAR

VAR
	tx :	TIME;
	last :	TIME;
	init :	BOOL;
	temp :	REAL;
	T_PLC_MS :	T_PLC_MS;
END_VAR

(*@KEY@: WORKSHEET
NAME: GEN_SIN
IEC_LANGUAGE: ST
*)
(* read system time and prepare input data *)
T_PLC_MS();
tx:= UDINT_TO_TIME(T_PLC_MS.T_PLC_MS) - last;

DL := modR(dl,1.0);
IF dl < 0.0 THEN dl := 1.0 - dl; END_IF;

(* init section *)
IF NOT init THEN
	init := TRUE;
	last := tx;
	tx := t#0s;
END_IF;

(* add last if one cycle is finished *)
IF tx >= pt THEN
	last := last + pt;
	tx := tx - pt;
END_IF;

(* generate sine wave *)
IF pt > t#0s THEN temp := SIN(6.283185307179586476 * TIME_TO_REAL(tx + multime(pt, dl)) / TIME_TO_REAL(pt)); END_IF;
out := am * 0.5 *  temp + os;

(* boolean output Q *)
q := NOT sign_R(temp);

(* revision history
hm	22. jan 2007	rev 1.0
	original version

hm	17 sep 2007	rev 1.1
	replaced time() with t_plc_ms for compatibilitx reasons

hm	27. nov 2007	rev 1.2
	avoid divide by 0 when pt = 0

hm	6. jan 2008		rev 1.3
	improved performance

hm	16. mar. 2008	rev 1.4
	added type conversion to avoid warnings under codesys 3.0

hm	18. oct. 2008	rev 1.5
	using math constants

hm	11. mar. 2009	rev 1.6
	changed real constants to use dot syntax

*)
(*@KEY@: END_WORKSHEET *)
END_FUNCTION_BLOCK

(* ---- GEN_SQ.ST ---- *)
(*@PROPERTIES_EX@
TYPE: POU
LOCALE: 0
IEC_LANGUAGE: ST
PLC_TYPE: independent
PROC_TYPE: independent
GROUP: LOGIC.GENERATORS
*)
(*@KEY@:DESCRIPTION*)
version 1.3	16. feb. 2011
programmer 	    hugo
tested by		tobias

gen_sq generates square wave signal with programmable period time.

(*@KEY@:END_DESCRIPTION*)
FUNCTION_BLOCK GEN_SQ

(*Group:Default*)

VAR_INPUT
	PT :	TIME;
END_VAR

VAR_OUTPUT
	Q :	BOOL;
END_VAR

VAR
	init :	BOOL;
	tn :	TIME;
	tx :	TIME;
	T_PLC_MS :	T_PLC_MS;
END_VAR

(*@KEY@: WORKSHEET
NAME: GEN_SQ
IEC_LANGUAGE: ST
*)
(* read system time *)
T_PLC_MS();
tx := UDINT_TO_TIME(T_PLC_MS.T_PLC_MS);

IF NOT init THEN
	init := TRUE;
	tn := tx;
	Q := TRUE;
ELSIF tx - tn >= DWORD_TO_TIME(SHR(TIME_TO_DWORD(PT),1)) THEN
	Q := NOT Q;
	tn := tn + DWORD_TO_TIME(SHR(TIME_TO_DWORD(pt),1));
END_IF;

(* revision history
hm	4. aug 2006	rev 1.0
	original version

hm	17. sep 2007	rev 1.1
	replaced time() with T_PLC_MS() for compatibility reasons

hm	18. jul. 2009	rev 1.2
	improved accuracy

hm	16. feb 2011	rev 1.3
	corrected an error with timer overflow
*)

(*@KEY@: END_WORKSHEET *)
END_FUNCTION_BLOCK

(* ---- GEN_SQR.ST ---- *)
(*@PROPERTIES_EX@
TYPE: POU
LOCALE: 0
IEC_LANGUAGE: ST
PLC_TYPE: independent
PROC_TYPE: independent
GROUP: ENGINEERING.SIGNAL_GENERATORS
*)
(*@KEY@:DESCRIPTION*)
version 1.4	11. mar. 2009
programmer 	oscat
tested BY	oscat

this signal generator generates a square wave output. The square wave signal is defined by period time (PT),
amplitude (AM), offset (OS), duty cycle (DC) and a specific delay for the output signal (DL).
The Output waveform will switch between AM/2 + OS and -AM/2 + OS. The DC input specifies ther duty cycle,
DC = 0 means output is low at all times and 1 means output is high at all times.
The delay input can delay a signal up to PT, this can be useful to synchronize different generators and generate interleaving signals.
in addition to a analog output Out there is a second boolean output Q.

(*@KEY@:END_DESCRIPTION*)
FUNCTION_BLOCK GEN_SQR

(*Group:Default*)

VAR_INPUT
	PT :	TIME;
	AM :	REAL := REAL#1.0;
	OS :	REAL;
	DC :	REAL := REAL#0.5;
	DL :	REAL;
END_VAR

VAR_OUTPUT
	Q :	BOOL;
	Out :	REAL;
END_VAR

VAR
	tx :	TIME;
	last :	TIME;
	init :	BOOL;
	T_PLC_MS :	T_PLC_MS;
END_VAR

(*@KEY@: WORKSHEET
NAME: GEN_SQR
IEC_LANGUAGE: ST
*)
(* check dc = 1 or 0 *)
IF dc = 0.0 THEN
	out := -am * 0.5 + os;
	Q := FALSE;
	RETURN;
ELSIF dc = 1.0 THEN
	out := am * 0.5 + os;
	Q := TRUE;
	RETURN;
END_IF;

(* read system time and prepare input data *)
T_PLC_MS();
tx:= UDINT_TO_TIME(T_PLC_MS.T_PLC_MS) - last;
DL := modR(dl,1.0);
IF dl < 0.0 THEN dl := 1.0 - dl; END_IF;
dc := modR(dc,1.0);
IF dc < 0.0 THEN dc := 1.0 - dc; END_IF;

(* init section *)
IF NOT init THEN
	init := TRUE;
	last := tx;
	tx := t#0s;
END_IF;

(* add last if one cycle is finished *)
IF tx >= pt THEN
	last := last + pt;
	tx := tx - pt;
END_IF;

(* check if falling or rising edge first *)
IF multime(pt, dl + dc) >= pt THEN
	(* generate falling edge *)
	IF tx >= multime(pt, dl + dc - 1.0) THEN
		out := -am * 0.5 + os;
		Q := FALSE;
	END_IF;
	(* generate rising edge *)
	IF tx >= multime(pt, dl) THEN
		out := am * 0.5 + os;
		Q := TRUE;
	END_IF;
ELSE
	(* generate rising edge first *)
	IF tx >= multime(pt, dl) THEN
		out := am * 0.5 + os;
		Q := TRUE;
	END_IF;
	(* generate falling edge *)
	IF tx >= multime(pt, dl + dc) THEN
		out := -am * 0.5 +os;
		Q := FALSE;
	END_IF;
END_IF;

(* revision history

hm	12. feb 2007	rev 1.1
	added default value for dc = 0.5

hm	17 sep 2007	rev 1.2
	replaced time() with t_plc_ms for compatibilitx reasons

hm	6. jan 2008	rev 1.3
	improved performance

hm	11. mar. 2009	rev 1.4
	changed real constants to use dot syntax
	set default amplitude to 1.0

*)

(*@KEY@: END_WORKSHEET *)
END_FUNCTION_BLOCK

(* ---- HEX_TO_BYTE.ST ---- *)
(*@PROPERTIES_EX@
TYPE: POU
LOCALE: 0
IEC_LANGUAGE: ST
PLC_TYPE: independent
PROC_TYPE: independent
GROUP: STRINGS
*)
(*@KEY@:DESCRIPTION*)
version 1.1	20. sep. 2008
programmer 	hugo
tested by		oscat

HEX_TO_BYTE converts a Hexadecimal string into a byte.
(*@KEY@:END_DESCRIPTION*)
FUNCTION_BLOCK HEX_TO_BYTE

(*Group:Default*)

VAR_INPUT
	HEX :	oscat_STRING5;
END_VAR

VAR_OUTPUT
	HEX_TO_BYTE :	BYTE;
END_VAR

VAR
	i :	INT;
	stop :	INT;
	X :	INT;
END_VAR

(*@KEY@: WORKSHEET
NAME: HEX_TO_BYTE
IEC_LANGUAGE: ST
*)
HEX_TO_BYTE := BYTE#0;
stop := LEN(HEX);
FOR I := 1 TO stop DO
	(* read the first character and subtract 48 to get value in decimal 0 = 48 *)
    x := GET_CHAR(Hex,I);
	(* calculate the value of the digit *)
	IF X > 47 AND x < 58 THEN
	    HEX_TO_BYTE := SHL_BYTE(HEX_TO_BYTE,4) OR INT_TO_BYTE (X - 48);
	ELSIF X > 64 AND X < 71 THEN
	    HEX_TO_BYTE := SHL_BYTE(HEX_TO_BYTE,4) OR INT_TO_BYTE (X - 55);
	ELSIF X > 96 AND X < 103 THEN
	    HEX_TO_BYTE := SHL_BYTE(HEX_TO_BYTE,4) OR INT_TO_BYTE (X - 87);
	END_IF;
END_FOR;

(* revision histroy
hm	18. jun. 2008	rev 1.0
	original release

hm	20. sep.2008	rev 1.1
	changed length of input string from 20 to 5

*)
(*@KEY@: END_WORKSHEET *)
END_FUNCTION_BLOCK

(* ---- HEX_TO_DWORD.ST ---- *)
(*@PROPERTIES_EX@
TYPE: POU
LOCALE: 0
IEC_LANGUAGE: ST
PLC_TYPE: independent
PROC_TYPE: independent
GROUP: STRINGS
*)
(*@KEY@:DESCRIPTION*)
version 1.4	18. jun. 2008
programmer 	hugo
tested by	tobias

HEX_TO_DWORD converts a Hexadecimal string into a DWORD.
(*@KEY@:END_DESCRIPTION*)
FUNCTION_BLOCK HEX_TO_DWORD

(*Group:Default*)

VAR_INPUT
	HEX :	oscat_STRING20;
END_VAR

VAR_OUTPUT
	HEX_TO_DWORD :	DWORD;
END_VAR

VAR
	i :	INT;
	stop :	INT;
	X :	INT;
END_VAR

(*@KEY@: WORKSHEET
NAME: HEX_TO_DWORD
IEC_LANGUAGE: ST
*)
HEX_TO_DWORD := DWORD#0;
stop := LEN(Hex);
FOR I := 1 TO stop DO
	(* read the first character and subtract 48 to get value in decimal 0 = 48 *)
    x := GET_CHAR(Hex,I);
	(* calculate the value of the digit *)
	IF X > 47 AND x < 58 THEN
	    HEX_TO_DWORD := SHL_DWORD(HEX_TO_DWORD,4) OR INT_TO_DWORD (X - 48);
	ELSIF X > 64 AND X < 71 THEN
	    HEX_TO_DWORD := SHL_DWORD(HEX_TO_DWORD,4) OR INT_TO_DWORD (X - 55);
	ELSIF X > 96 AND X < 103 THEN
	    HEX_TO_DWORD := SHL_DWORD(HEX_TO_DWORD,4) OR INT_TO_DWORD (X - 87);
	END_IF;
END_FOR;

(* revision histroy
hm	2.10.2007		rev 1.0
	original release

hm	19.11.2007		rev 1.1
	changed type of function from int to dword

hm 	4. mar 2008		rev 1.2
	added support for a..f and return 0 for invalid string

hm	29. mar. 2008	rev 1.3
	changed STRING to STRING(8)

hm	18. jun. 2008	rev 1.4
	changed input hex to STRING(20)
	function now ignores wrong characters
*)
(*@KEY@: END_WORKSHEET *)
END_FUNCTION_BLOCK

(* ---- HOLIDAY.ST ---- *)
(*@PROPERTIES_EX@
TYPE: POU
LOCALE: 0
IEC_LANGUAGE: ST
PLC_TYPE: independent
PROC_TYPE: independent
GROUP: TIME_DATE
*)
(*@KEY@:DESCRIPTION*)
version 2.0	18. jans 2011
programmer 	hugo
tested by	tobias

holiday calculates if a given day is a holiday and displays the name of the holiday as string as well as a boolean flag to indicate a holiday.
the holidays are specified in the country setup under global constants.
a holiday can be of fixed date for example new years day on january 1st.
a holiday can have a fixed offset from easter sunday as for most church holidays.
a holiday can be a specific weekday before a fixed date, for example buss und bettag is the last wednesday before nov 23rd.
with a simple f_use flag any specific holiday can be turned on or off if needed.

please check the manual for examples of holiday definitions

(*@KEY@:END_DESCRIPTION*)
FUNCTION_BLOCK HOLIDAY

(*Group:Parameter*)

VAR_INPUT
	DATE_IN :	UDINT;
	LANGU :	INT;
	FRIDAY :	BOOL;
	SATURDAY :	BOOL;
	SUNDAY :	BOOL;
END_VAR

VAR_OUTPUT
	Y :	BOOL;
	NAME :	oscat_STRING30;
END_VAR

VAR_IN_OUT
	HOLIDAYS :	oscat_HOLIDAY_DATA_0_29;
END_VAR

(*Group:lokal*)

VAR
	size :	INT := INT#29;
	last_active :	UDINT;
	ostern :	UDINT;
	i :	INT;
	jahr :	INT;
	x_date :	UDINT;
	lx :	INT;
	wdx :	INT;
	SETUP_LOCATION :	SETUP_LOCATION;
	SETUP_WEEKDAYS :	SETUP_WEEKDAYS;
	SETUP_LANGUAGE :	SETUP_LANGUAGE;
	LOCATION :	oscat_LOCATION;
	WEEKDAYS :	oscat_WEEKDAYS;
	LANGUAGE :	oscat_LANGUAGE;
	wd :	INT;
END_VAR

(*@KEY@: WORKSHEET
NAME: HOLIDAY
IEC_LANGUAGE: ST
*)
(* for performance reasons only activate once a day *)
IF last_active = date_in THEN RETURN; END_IF;
last_active := DATE_IN;

SETUP_LOCATION(LOCATION:=LOCATION);
LOCATION:=SETUP_LOCATION.LOCATION;

SETUP_WEEKDAYS(WEEKDAYS:=WEEKDAYS);
WEEKDAYS:=SETUP_WEEKDAYS.WEEKDAYS;

SETUP_LANGUAGE(LANGUAGE:=LANGUAGE);
LANGUAGE:=SETUP_LANGUAGE.LANGUAGE;

(* determine language *)
IF LANGU = 0 THEN
	lx := language.DEFAULT;
ELSE
	lx := MIN(language.LMAX, LANGU);
END_IF;

(* berechnung von ostern für das aktuelle jahr *)
jahr := YEAR_OF_DATE(date_in);
ostern := EASTER(jahr);
wdx := DAY_OF_WEEK(DATE_IN);
Y := FALSE;

(* check for holidays *)
FOR i := 0 TO size DO
	x_date := SET_DATE(jahr, SINT_TO_INT(HOLIDAYS[i].MONTH) , SINT_TO_INT(HOLIDAYS[i].DAY));
	IF HOLIDAYS[i].USE = SINT#1 AND HOLIDAYS[i].MONTH > SINT#0 THEN
		(* check for fixed date holiday *)
		IF x_date = date_in THEN
			Y := TRUE;
			NAME := HOLIDAYS[i].NAME;
			RETURN;
		END_IF;
	ELSIF HOLIDAYS[i].USE = SINT#1 AND HOLIDAYS[i].MONTH = SINT#0 THEN
		(* check for holiday in reference to easter *)
		IF DATE_ADD(ostern, SINT_TO_INT(HOLIDAYS[i].DAY),0,0,0) = date_in THEN
			Y := TRUE;
			NAME := HOLIDAYS[i].NAME;
			RETURN;
		END_IF;
	ELSIF HOLIDAYS[i].USE < SINT#0 THEN
		(* check for holiday on a weekday before date *)
		IF DAY_OF_WEEK(date_in) = SINT_TO_INT(ABS(HOLIDAYS[i].USE)) AND date_in < x_date AND date_in >= DATE_ADD(x_date,-7,0,0,0) THEN
			Y := TRUE;
			NAME := HOLIDAYS[i].NAME;
			RETURN;
		END_IF;
	END_IF;
END_FOR;

(* check array if today is weekend *)
IF NOT Y AND (wdx = 5 AND FRIDAY OR wdx = 6 AND SATURDAY OR wdx = 7 AND SUNDAY) THEN
	Y := TRUE;
	wd := LOCATION.LANGUAGE[lx];
	NAME := WEEKDAYS[wd][wdx];
ELSE
	NAME := '';
END_IF;

(*
Neujahrstag 	1. Januar 	• 	• 	• 	• 	• 	• 	• 	• 	• 	• 	• 	• 	• 	• 	• 	•
Heilige Drei Könige 	6. Januar 	• 	• 												•
Karfreitag 	Ostersonntag - 2d 	• 	• 	• 	• 	• 	• 	• 	• 	• 	• 	• 	• 	• 	• 	• 	•
Ostersonntag 	siehe Osterdatum 				(•)
Ostermontag 	Ostersonntag + 1d 	• 	• 	• 	• 	• 	• 	• 	• 	• 	• 	• 	• 	• 	• 	• 	•
Tag der Arbeit 	1. Mai 	• 	• 	• 	• 	• 	• 	• 	• 	• 	• 	• 	• 	• 	• 	• 	•
Christi Himmelfahrt 	Ostersonntag + 39d 	• 	• 	• 	• 	• 	• 	• 	• 	• 	• 	• 	• 	• 	• 	• 	•
Pfingstsonntag 	Ostersonntag + 49d 				(•)
Pfingstmontag 	Ostersonntag + 50d 	• 	• 	• 	• 	• 	• 	• 	• 	• 	• 	• 	• 	• 	• 	• 	•
Fronleichnam 	Ostersonntag + 60d 	• 	• 					• 			• 	• 	• 	1) 			2)
Augsburger Friedensfest 	8. August 		(3)
Mariä Himmelfahrt 	15. August 		(5) 										•
Tag der Deutschen Einheit 	3. Oktober 6) 	• 	• 	• 	• 	• 	• 	• 	• 	• 	• 	• 	• 	• 	• 	• 	•
Reformationstag 	31. Oktober 				• 				• 					• 	• 		•
Allerheiligen 	1. November 	• 	• 								• 	• 	•
Buß- und Bettag 4) 	Mittwoch vor dem 23.11. 			7 										•
1. Weihnachtstag 	25. Dezember 	• 	• 	• 	• 	• 	• 	• 	• 	• 	• 	• 	• 	• 	• 	• 	•
2. Weihnachtstag 	26. Dezember 	• 	• 	• 	• 	• 	• 	• 	• 	• 	• 	• 	• 	• 	• 	• 	•
*)

(* revision history
hm 	27. feb. 2007	rev 1.1
	deleted unused variable init

hm	31. oct. 2007	rev 1.2
	changed holiday definition from constant to input constant to allow easier changes by user without recompilation of the lib

hm 	24. nov. 2007	rev 1.3
	changes F_use of  Buß_und_Bettag to 0 because this is no official holiday

hm	7. apr. 2008	rev 1.4
	improved performance

hm	7. oct. 2008	rev 1.5
	changed code to use setup data from global constants
	changed length of output NAME from 20 to 30
	holiday will now also be indicated on a weekend
	changed function year to year_of_date
	changed function weekday to day_of_week

hm	21. oct. 2008	rev 1.6
	using location constants

hm	18. jan 2011	rev 2.0
	using user specified array for holidays

*)

(*@KEY@: END_WORKSHEET *)
END_FUNCTION_BLOCK

(* ---- HYST.ST ---- *)
(*@PROPERTIES_EX@
TYPE: POU
LOCALE: 0
IEC_LANGUAGE: ST
PLC_TYPE: independent
PROC_TYPE: independent
GROUP: ENGINEERING.CONTROL
*)
(*@KEY@:DESCRIPTION*)
version 1.0	2. jun. 2008
programmer 	hugo
tested BY	tobias

This Hystereses function has two modes:
1. if on > off then Q will be switched high when in > on and switched low when in < off.
2. if on < off then Q will be switched high when in < on and switched low when in > off.
the output win will be high when in is between low and high.
(*@KEY@:END_DESCRIPTION*)
FUNCTION_BLOCK HYST

(*Group:Default*)

VAR_INPUT
	IN :	REAL;
	ON :	REAL;
	OFF :	REAL;
END_VAR

VAR_OUTPUT
	Q :	BOOL;
	WIN :	BOOL;
END_VAR

(*@KEY@: WORKSHEET
NAME: HYST
IEC_LANGUAGE: ST
*)
IF ON >= OFF THEN
	IF IN < OFF THEN
		Q := FALSE;
		WIN := FALSE;
	ELSIF  IN > ON THEN
		Q := TRUE;
		WIN := FALSE;
	ELSE
		WIN := TRUE;
	END_IF;
ELSE
	IF IN > OFF THEN
		Q := FALSE;
		WIN := FALSE;
	ELSIF  IN < ON THEN
		Q := TRUE;
		WIN := FALSE;
	ELSE
		WIN := TRUE;
	END_IF;
END_IF;

(* revision history
hm		2.  jun 2008	rev 1.0
	original version

*)
(*@KEY@: END_WORKSHEET *)
END_FUNCTION_BLOCK

(* ---- HYST_1.ST ---- *)
(*@PROPERTIES_EX@
TYPE: POU
LOCALE: 0
IEC_LANGUAGE: ST
PLC_TYPE: independent
PROC_TYPE: independent
GROUP: ENGINEERING.CONTROL
*)
(*@KEY@:DESCRIPTION*)
version 1.1	2. jun. 2008
programmer 	hugo
tested BY	tobias

this hysteresis function switches the output high if the input signal reaches obove high and will switch to low when the input falls back below low value.
a separate output mid is set if the input stays between low and high value.
(*@KEY@:END_DESCRIPTION*)
FUNCTION_BLOCK HYST_1

(*Group:Default*)

VAR_INPUT
	IN :	REAL;
	HIGH :	REAL;
	LOW :	REAL;
END_VAR

VAR_OUTPUT
	Q :	BOOL;
	WIN :	BOOL;
END_VAR

(*@KEY@: WORKSHEET
NAME: HYST_1
IEC_LANGUAGE: ST
*)
IF in < low THEN
	Q := FALSE;
	win := FALSE;
ELSIF in > high THEN
	Q := TRUE;
	win := FALSE;
ELSE
	win := TRUE;
END_IF;

(* code used for rev 1.0
IF Q THEN
	IF in < low THEN q := FALSE; END_IF;
ELSE
	IF in > high THEN q := TRUE; END_IF;
END_IF;
win := in > low AND in < high;
*)
(*@KEY@: END_WORKSHEET *)
END_FUNCTION_BLOCK

(* ---- HYST_2.ST ---- *)
(*@PROPERTIES_EX@
TYPE: POU
LOCALE: 0
IEC_LANGUAGE: ST
PLC_TYPE: independent
PROC_TYPE: independent
GROUP: ENGINEERING.CONTROL
*)
(*@KEY@:DESCRIPTION*)
version 1.2	2. jun. 2008
programmer 	oscat
tested BY	tobias

this hysteresis function switches the output high if the input signal reaches obove val + hys/2 and will switch to low when the input falls back below val - hys/2 value.
a separate output mid is set if the input stays between low and high value.
(*@KEY@:END_DESCRIPTION*)
FUNCTION_BLOCK HYST_2

(*Group:Default*)

VAR_INPUT
	IN :	REAL;
	VAL :	REAL;
	HYS :	REAL;
END_VAR

VAR_OUTPUT
	Q :	BOOL;
	WIN :	BOOL;
END_VAR

VAR
	tmp :	REAL;
END_VAR

(*@KEY@: WORKSHEET
NAME: HYST_2
IEC_LANGUAGE: ST
*)
tmp := val - hys * 0.5;
IF in < tmp THEN
	Q := FALSE;
	win := FALSE;
ELSIF in > tmp + hys THEN
	Q := TRUE;
	win := FALSE;
ELSE
	win := TRUE;
END_IF;

(* code used for 1.2 and before
X := hys * 0.5;
IF Q THEN
	IF in < val - x THEN q := FALSE; END_IF;
ELSE
	IF in > val + x THEN q := TRUE; END_IF;
END_IF;
win := in > val - x AND in < val + x;
*)

(* revision history
hm		4. aug 2006	rev 1.0
	original version

hm		5. jan 2008	rev 1.1
	improved code for better performance

hm		2. jun. 2008	rev 1.2
	improved performance
*)
(*@KEY@: END_WORKSHEET *)
END_FUNCTION_BLOCK

(* ---- HYST_3.ST ---- *)
(*@PROPERTIES_EX@
TYPE: POU
LOCALE: 0
IEC_LANGUAGE: ST
PLC_TYPE: independent
PROC_TYPE: independent
GROUP: ENGINEERING.CONTROL
*)
(*@KEY@:DESCRIPTION*)
version 1.2	5 jan 2008
programmer 	oscat
tested BY	tobias

this is a double hysteresis function. Out1 follows a hysteresis function defined by val1and hyst, while out 2 follows val2 and hyst.
if the input signal is between the two hysteresis switches (val1 and val2) then non of the outputs is active.
(*@KEY@:END_DESCRIPTION*)
FUNCTION_BLOCK HYST_3

(*Group:Default*)

VAR_INPUT
	IN :	REAL;
	HYST :	REAL;
	VAL1 :	REAL;
	VAL2 :	REAL;
END_VAR

VAR_OUTPUT
	Q1 :	BOOL;
	Q2 :	BOOL;
END_VAR

VAR
	X :	REAL;
END_VAR

(*@KEY@: WORKSHEET
NAME: HYST_3
IEC_LANGUAGE: ST
*)
X := hyst * 0.5;
IF in < val1 - X THEN
	q1 := TRUE;
ELSIF in > val1 + X THEN
	q1 := FALSE;
END_IF;
IF in < val2 - X THEN
	q2 := FALSE;
ELSIF in > val2 + X THEN
	q2 := TRUE;
END_IF;

(* revision history
hm	22. jan 2007	rev 1.0
	original version

hm	27. dec 2007	rev 1.1
	changed code for better performance

hm	5. jan 2008		rev 1.2
	further performance iprovements

*)
(*@KEY@: END_WORKSHEET *)
END_FUNCTION_BLOCK

(* ---- INC_DEC.ST ---- *)
(*@PROPERTIES_EX@
TYPE: POU
LOCALE: 0
IEC_LANGUAGE: ST
PLC_TYPE: independent
PROC_TYPE: independent
GROUP: ENGINEERING.AUTOMATION
*)
(*@KEY@:DESCRIPTION*)
version 1.0	4 aug 2006
programmer 	oscat
tested BY	oscat

incremental decoder with quadruple accuracy.
2 pulses for each channel are created for each directional pulse.
(*@KEY@:END_DESCRIPTION*)
FUNCTION_BLOCK INC_DEC

(*Group:Default*)

VAR_INPUT
	CHA :	BOOL;
	CHB :	BOOL;
	RST :	BOOL := 0;
END_VAR

VAR_OUTPUT
	DIR :	BOOL;
	CNT :	INT;
END_VAR

VAR
	edgea :	BOOL := 0;
	clk :	BOOL;
	clka :	BOOL;
	clkb :	BOOL;
	edgeb :	BOOL;
	axb :	BOOL;
END_VAR

(*@KEY@: WORKSHEET
NAME: INC_DEC
IEC_LANGUAGE: ST
*)
axb := cha XOR chb;

(* create pulses for channel a *)
clka := cha XOR edgea;
edgea := cha;

clkb := chb XOR edgeb;
edgeb := chb;

(* create pulses for both channels *)
clk := clka OR clkb;

(* set the direction output *)
IF axb AND clka THEN dir := TRUE; END_IF;
IF axb AND clkb THEN dir := FALSE; END_IF;

(* increment or decrement the counter *)
IF clk AND dir THEN cnt := cnt + 1; END_IF;
IF clk AND NOT dir THEN cnt := cnt -1; END_IF;

(* reset the counter if rst active *)
IF rst THEN cnt := 0; END_IF;
(*@KEY@: END_WORKSHEET *)
END_FUNCTION_BLOCK

(* ---- INTEGRATE.ST ---- *)
(*@PROPERTIES_EX@
TYPE: POU
LOCALE: 0
IEC_LANGUAGE: ST
PLC_TYPE: independent
PROC_TYPE: independent
GROUP: ENGINEERING.CONTROL
*)
(*@KEY@:DESCRIPTION*)
version 1.0	3. nov. 2008
programmer 	hugo
tested by	oscat

integrate is a plain integrator with I/O for out.
(*@KEY@:END_DESCRIPTION*)
FUNCTION_BLOCK INTEGRATE

(*Group:Default*)

VAR_INPUT
	E :	BOOL := TRUE;
	X :	REAL;
	K :	REAL := 1.0;
END_VAR

VAR_IN_OUT
	Y :	REAL;
END_VAR

VAR
	X_last :	REAL;
	init :	BOOL;
	T_PLC_MS :	T_PLC_MS;
	last :	UDINT;
	tx :	UDINT;
END_VAR

(*@KEY@: WORKSHEET
NAME: INTEGRATE
IEC_LANGUAGE: ST
*)
(* read system time *)
T_PLC_MS();
tx:= T_PLC_MS.T_PLC_MS;

IF NOT init THEN
	init := TRUE;
	X_last := X;
ELSIF E THEN
	Y := (X + X_LAST) * 0.5E-3 * UDINT_TO_REAL(tx-last) * K + Y;
	X_last := X;
END_IF;
last := tx;

(*
hm 	3. nov. 2008	rev 1.0
original version

*)
(*@KEY@: END_WORKSHEET *)
END_FUNCTION_BLOCK

(* ---- INTERLOCK.ST ---- *)
(*@PROPERTIES_EX@
TYPE: POU
LOCALE: 0
IEC_LANGUAGE: ST
PLC_TYPE: independent
PROC_TYPE: independent
GROUP: ENGINEERING.AUTOMATION
*)
(*@KEY@:DESCRIPTION*)
version 1.0	28 sep 2007
programmer 	hugo
tested by	tobias

INTERLOCK has two inputs I1 and I2 which drive the corresponding outputs Q1 and Q2.
the inputs signals lock each other out and therfore I1 can only drive Q1 when I2 is Low and vice versa.
The input TL specifies a dead time between two outputs can become active.
an output can only become active when the other output was not active for the time TL.
(*@KEY@:END_DESCRIPTION*)
FUNCTION_BLOCK INTERLOCK

(*Group:Default*)

VAR_INPUT
	I1 :	BOOL;
	I2 :	BOOL;
	TL :	TIME;
END_VAR

VAR_OUTPUT
	Q1 :	BOOL;
	Q2 :	BOOL;
END_VAR

VAR
	T1 :	TOF;
	T2 :	TOF;
END_VAR

(*@KEY@: WORKSHEET
NAME: INTERLOCK
IEC_LANGUAGE: ST
*)
(* the input signal have a run delay to lockout the other input *)
T1(IN := I1, PT := TL);
T2(IN := I2, PT := TL);

Q1 := I1 AND NOT t2.Q;
Q2 := I2 AND NOT t1.Q;

(* revision history

hm	28 sep 2007		rev 1.0
	original version

*)
(*@KEY@: END_WORKSHEET *)
END_FUNCTION_BLOCK

(* ---- INTERLOCK_4.ST ---- *)
(*@PROPERTIES_EX@
TYPE: POU
LOCALE: 0
IEC_LANGUAGE: ST
PLC_TYPE: independent
PROC_TYPE: independent
GROUP: ENGINEERING.AUTOMATION
*)
(*@KEY@:DESCRIPTION*)
version 1.1	14. mar. 2009
programmer 	hugo
tested by	oscat

INTERLOCK_4 detects one of 4 switches and delivers the number of the switch pressed on the output out
a output tp is true for one cycle if the output has changed.
a setup variable MODE selects between 3 different modes:
MODE = 0, any input active will disable all other inputs
MODE = 1, the input with the highest number will be acepted
mode = 2, the input last pressed will disable all others

(*@KEY@:END_DESCRIPTION*)
FUNCTION_BLOCK INTERLOCK_4

(*Group:Default*)

VAR_INPUT
	I0 :	BOOL;
	I1 :	BOOL;
	I2 :	BOOL;
	I3 :	BOOL;
	E :	BOOL;
	MODE :	INT;
END_VAR

VAR_OUTPUT
	OUT :	BYTE;
	TP :	BOOL;
END_VAR

VAR
	in :	BYTE;
	last :	BYTE;
	old :	BYTE;
	lmode :	INT;
END_VAR

(*@KEY@: WORKSHEET
NAME: INTERLOCK_4
IEC_LANGUAGE: ST
*)
(* check if enable is active *)
IF E THEN
(* reset all vars when there is a mode change on thy fly *)
	IF mode <> lmode THEN
		out := BYTE#0;
		last := BYTE#0;
		old := BYTE#0;
		lmode := mode;
	END_IF;
	(* load inputs into in *)
	in:=BIT_LOAD_B(in,I0,0); (* in.0 *)
	in:=BIT_LOAD_B(in,I1,1); (* in.1 *)
	in:=BIT_LOAD_B(in,I2,2); (* in.2 *)
	in:=BIT_LOAD_B(in,I3,3); (* in.3 *)
	(* only execute when there is any change *)
	IF in <> last THEN
		(* only execute when inputs have chages state *)
		CASE mode OF
			0:	(* output directly display inputs as bits in byte out *)
				out := in;

			1:	(* the input with the highest number will be acepted *)
				IF    (in AND BYTE#2#00001000) > BYTE#0 (* in.3 *) THEN out := BYTE#8;
				ELSIF (in AND BYTE#2#00000100) > BYTE#0 (* in.2 *) THEN out := BYTE#4;
				ELSIF (in AND BYTE#2#00000010) > BYTE#0 (* in.1 *) THEN out := BYTE#2;
				ELSE out := in;
				END_IF;

			2:	(* input last pressed will be displayed only *)
				last := ((in XOR last) AND in);
				IF    (last AND BYTE#2#00001000) > BYTE#0 (* last.3 *) THEN out := BYTE#8;
				ELSIF (last AND BYTE#2#00000100) > BYTE#0 (* last.2 *) THEN out := BYTE#4;
				ELSIF (last AND BYTE#2#00000010) > BYTE#0 (* last.1 *) THEN out := BYTE#2;
				ELSE out := last;
				END_IF;

			3:	(* any input active will disable all other inputs *)
				IF (out AND in) = BYTE#0 THEN
					IF    (in AND BYTE#2#00001000) > BYTE#0 (* in.3 *) THEN out := BYTE#8;
					ELSIF (in AND BYTE#2#00000100) > BYTE#0 (* in.2 *) THEN out := BYTE#4;
					ELSIF (in AND BYTE#2#00000010) > BYTE#0 (* in.1 *) THEN out := BYTE#2;
					ELSE out := in;
					END_IF;
				END_IF;

		END_CASE;
		last := in;
	END_IF;
	tp := out <> old;
	old := out;
ELSE
	out := BYTE#0;
	last := BYTE#0;
	old := BYTE#0;
	lmode := 0;
	tp := FALSE;
END_IF;

(* revision history
hm	24. oct 2008	rev 1.0
	original version

hm	14. mar. 2009	rev 1.1
	replaced double assignments

*)
(*@KEY@: END_WORKSHEET *)
END_FUNCTION_BLOCK

(* ---- IS_ALNUM.ST ---- *)
(*@PROPERTIES_EX@
TYPE: POU
LOCALE: 0
IEC_LANGUAGE: ST
PLC_TYPE: independent
PROC_TYPE: independent
GROUP: STRINGS
*)
(*@KEY@:DESCRIPTION*)
version 1.1	29. mar. 2008
programmer 		kurt
tested by		hugo

ISC_ALNUM testet ob in einem string nur Zahlen 0..9 vorkommen.
(*@KEY@:END_DESCRIPTION*)
FUNCTION_BLOCK IS_ALNUM

(*Group:Default*)

VAR_INPUT
	STR :	STRING;
END_VAR

VAR_OUTPUT
	IS_ALNUM :	BOOL;
END_VAR

VAR
	char :	BYTE;
	pos :	INT;
	I :	INT;
END_VAR

(*@KEY@: WORKSHEET
NAME: IS_ALNUM
IEC_LANGUAGE: ST
*)
I := LEN(str);
FOR pos := 1 TO I DO
    char := INT_TO_BYTE(GET_CHAR(str,pos));
	IF NOT (ISC_ALPHA(char) OR ISC_NUM(char)) THEN
		IS_ALNUM := FALSE;
		RETURN;
	END_IF;
END_FOR;
IS_ALNUM := I<>0;

(* revision history
hm	29. feb 2008	rev 1.0
	original version

hm	29. mar. 2008	rev 1.1
	changed STRING to STRING(STRING_LENGTH)
*)
(*@KEY@: END_WORKSHEET *)
END_FUNCTION_BLOCK

(* ---- IS_ALPHA.ST ---- *)
(*@PROPERTIES_EX@
TYPE: POU
LOCALE: 0
IEC_LANGUAGE: ST
PLC_TYPE: independent
PROC_TYPE: independent
GROUP: STRINGS
*)
(*@KEY@:DESCRIPTION*)
version 1.1	29. mar. 2008
programmer 		kurt
tested by		hugo

IS_ALPHA testet ob in einem string nur Zeichen a-z oder A - Z vorkommen.
(*@KEY@:END_DESCRIPTION*)
FUNCTION_BLOCK IS_ALPHA

(*Group:Default*)

VAR_INPUT
	STR :	STRING;
END_VAR

VAR_OUTPUT
	IS_ALPHA :	BOOL;
END_VAR

VAR
	pos :	INT;
	I :	INT;
END_VAR

(*@KEY@: WORKSHEET
NAME: IS_ALPHA
IEC_LANGUAGE: ST
*)
I := LEN(str);
FOR pos := 1 TO I DO
	IF NOT ISC_ALPHA(INT_TO_BYTE(GET_CHAR(str,pos))) THEN
		IS_ALPHA := FALSE;
		RETURN;
	END_IF;
END_FOR;
IS_ALPHA := NOT (I=0);

(* revision history
hm	29. feb 2008	rev 1.0
	original version

hm	29. mar. 2008	rev 1.1
	changed STRING to STRING(STRING_LENGTH)
*)
(*@KEY@: END_WORKSHEET *)
END_FUNCTION_BLOCK

(* ---- IS_CC.ST ---- *)
(*@PROPERTIES_EX@
TYPE: POU
LOCALE: 0
IEC_LANGUAGE: ST
PLC_TYPE: independent
PROC_TYPE: independent
GROUP: STRINGS
*)
(*@KEY@:DESCRIPTION*)
version 1.1	29. mar. 2008
programmer 	Tobias
tested by	hugo

ISC_CC testet ob ein string nur aus Zeichen des Strings CMP besteht.
(*@KEY@:END_DESCRIPTION*)
FUNCTION_BLOCK IS_CC

(*Group:Default*)

VAR_INPUT
	STR :	STRING;
	CMP :	STRING;
END_VAR

VAR_OUTPUT
	IS_CC :	BOOL;
END_VAR

VAR
	L :	INT;
	pos :	INT;
	temp :	STRING;
END_VAR

(*@KEY@: WORKSHEET
NAME: IS_CC
IEC_LANGUAGE: ST
*)
L := LEN(str);
FOR pos := 1 TO L DO
    temp := MID(str,1,pos);
	IF FIND(CMP,temp) = 0 THEN
	    IS_CC := FALSE;
	    RETURN;
	END_IF;
END_FOR;
IS_CC := L > 0;

(* revision history
hm	19. mar 2008	rev 1.0
	original version

hm	29. mar. 2008	rev 1.1
	changed STRING to STRING(STRING_LENGTH)
*)
(*@KEY@: END_WORKSHEET *)
END_FUNCTION_BLOCK

(* ---- IS_CTRL.ST ---- *)
(*@PROPERTIES_EX@
TYPE: POU
LOCALE: 0
IEC_LANGUAGE: ST
PLC_TYPE: independent
PROC_TYPE: independent
GROUP: STRINGS
*)
(*@KEY@:DESCRIPTION*)
version 1.1	29. mar 2008
programmer 		kurt
tested by		hugo

IS_CTRL testet ob in einem string nur Steuerzeichen (Char < 32) vorkommen.
(*@KEY@:END_DESCRIPTION*)
FUNCTION_BLOCK IS_CTRL

(*Group:Default*)

VAR_INPUT
	STR :	STRING;
END_VAR

VAR_OUTPUT
	IS_CTRL :	BOOL;
END_VAR

VAR
	pos :	INT;
	I :	INT;
END_VAR

(*@KEY@: WORKSHEET
NAME: IS_CTRL
IEC_LANGUAGE: ST
*)
I := LEN(str);
FOR pos := 1 TO I DO
	IF NOT ISC_CTRL(INT_TO_BYTE(GET_CHAR(str,pos))) THEN
		IS_CTRL := FALSE;
		RETURN;
	END_IF;
END_FOR;
IS_CTRL := I > 0;

(* revision history
hm	29. feb. 2008	rev 1.0
	original version

hm	29. mar. 2008	rev 1.1
	changed STRING to STRING(STRING_LENGTH)
*)
(*@KEY@: END_WORKSHEET *)
END_FUNCTION_BLOCK

(* ---- IS_HEX.ST ---- *)
(*@PROPERTIES_EX@
TYPE: POU
LOCALE: 0
IEC_LANGUAGE: ST
PLC_TYPE: independent
PROC_TYPE: independent
GROUP: STRINGS
*)
(*@KEY@:DESCRIPTION*)
version 1.1	29. mar. 2008
programmer 		kurt
tested by		hugo

IS_HEX testet ob in einem string nur Zahlen 0..9 oder A..F oder a..f  vorkommen.
(*@KEY@:END_DESCRIPTION*)
FUNCTION_BLOCK IS_HEX

(*Group:Default*)

VAR_INPUT
	STR :	STRING;
END_VAR

VAR_OUTPUT
	IS_HEX :	BOOL;
END_VAR

VAR
	pos :	INT;
	I :	INT;
END_VAR

(*@KEY@: WORKSHEET
NAME: IS_HEX
IEC_LANGUAGE: ST
*)
I := LEN(str);
FOR pos := 1 TO I DO
	IF NOT ISC_HEX(INT_TO_BYTE(GET_CHAR(str,pos))) THEN
		IS_HEX := FALSE;
		RETURN;
	END_IF;
END_FOR;
IS_HEX := I>0;

(* revision history
hm	29. feb 2008	rev 1.0
	original version

hm	29. mar. 2008	rev 1.1
	changed STRING to STRING(STRING_LENGTH)
*)
(*@KEY@: END_WORKSHEET *)
END_FUNCTION_BLOCK

(* ---- IS_LOWER.ST ---- *)
(*@PROPERTIES_EX@
TYPE: POU
LOCALE: 0
IEC_LANGUAGE: ST
PLC_TYPE: independent
PROC_TYPE: independent
GROUP: STRINGS
*)
(*@KEY@:DESCRIPTION*)
version 1.1	29. mar. 2008
programmer 		kurt
tested by		hugo

IS_LOWER testet ob in einem string nur kleinbuchstaben vorkommen.
(*@KEY@:END_DESCRIPTION*)
FUNCTION_BLOCK IS_LOWER

(*Group:Default*)

VAR_INPUT
	STR :	STRING;
END_VAR

VAR_OUTPUT
	IS_LOWER :	BOOL;
END_VAR

VAR
	pos :	INT;
	I :	INT;
END_VAR

(*@KEY@: WORKSHEET
NAME: IS_LOWER
IEC_LANGUAGE: ST
*)
I := LEN(str);
FOR pos := 1 TO I DO
	IF NOT ISC_LOWER(INT_TO_BYTE(GET_CHAR(str,pos))) THEN
		IS_LOWER := FALSE;
		RETURN;
	END_IF;
END_FOR;
IS_LOWER := I>0;

(* revision history
hm	29. feb 2008	rev 1.0
	original version

hm	29. mar. 2008	rev 1.1
	changed STRING to STRING(STRING_LENGTH)
*)
(*@KEY@: END_WORKSHEET *)
END_FUNCTION_BLOCK

(* ---- IS_NCC.ST ---- *)
(*@PROPERTIES_EX@
TYPE: POU
LOCALE: 0
IEC_LANGUAGE: ST
PLC_TYPE: independent
PROC_TYPE: independent
GROUP: STRINGS
*)
(*@KEY@:DESCRIPTION*)
version 1.1	29. mar. 2008
programmer 		Tobias
tested by		hugo

ISC_NCC testet ob in einem string keine Zeichen des Strings CMP enthalten sind.
(*@KEY@:END_DESCRIPTION*)
FUNCTION_BLOCK IS_NCC

(*Group:Default*)

VAR_INPUT
	STR :	STRING;
	CMP :	STRING;
END_VAR

VAR_OUTPUT
	IS_NCC :	BOOL;
END_VAR

VAR
	L :	INT;
	pos :	INT;
	temp :	STRING;
END_VAR

(*@KEY@: WORKSHEET
NAME: IS_NCC
IEC_LANGUAGE: ST
*)
L := LEN(str);
FOR pos := 1 TO L DO
    temp := MID(str,1,pos);
	IF FIND(CMP,temp) > 0 THEN
	    IS_NCC := FALSE;
	    RETURN;
	END_IF;
END_FOR;
IS_NCC := TRUE;

(* revision history
hm	19. mar 2008	rev 1.0
	original version

hm	29. mar. 2008	rev 1.1
	changed STRING to STRING(STRING_LENGTH)
*)
(*@KEY@: END_WORKSHEET *)
END_FUNCTION_BLOCK

(* ---- IS_NUM.ST ---- *)
(*@PROPERTIES_EX@
TYPE: POU
LOCALE: 0
IEC_LANGUAGE: ST
PLC_TYPE: independent
PROC_TYPE: independent
GROUP: STRINGS
*)
(*@KEY@:DESCRIPTION*)
version 1.1	29. mar. 2008
programmer 		kurt
tested by		hugo

IS_NUM testet ob in einem string nur Zahlen 0..9 vorkommen.
(*@KEY@:END_DESCRIPTION*)
FUNCTION_BLOCK IS_NUM

(*Group:Default*)

VAR_INPUT
	STR :	STRING;
END_VAR

VAR_OUTPUT
	IS_NUM :	BOOL;
END_VAR

VAR
	pos :	INT;
	I :	INT;
END_VAR

(*@KEY@: WORKSHEET
NAME: IS_NUM
IEC_LANGUAGE: ST
*)
I := LEN(str);
FOR pos := 1 TO I DO
	IF NOT ISC_NUM(INT_TO_BYTE(GET_CHAR(str,pos))) THEN
		IS_NUM := FALSE;
		RETURN;
	END_IF;
END_FOR;
IS_NUM := I>0;

(* revision history
hm	29. feb 2008	rev 1.0
	original version

hm	29. mar. 2008	rev 1.1
	changed STRING to STRING(STRING_LENGTH)
*)
(*@KEY@: END_WORKSHEET *)
END_FUNCTION_BLOCK

(* ---- IS_SORTED.ST ---- *)
(*@PROPERTIES_EX@
TYPE: POU
LOCALE: 0
IEC_LANGUAGE: ST
PLC_TYPE: independent
PROC_TYPE: independent
GROUP: MATHEMATICAL.ARRAY_FUNCTIONS
*)
(*@KEY@:DESCRIPTION*)
version 1.1	4. apr. 2008
programmer 	hugo
tested by	tobias

this function will return true if the given array is sorted in an ascending order.
(*@KEY@:END_DESCRIPTION*)
FUNCTION_BLOCK IS_SORTED

(*Group:Default*)

VAR_IN_OUT
	PT :	oscat_pt_ARRAY;
END_VAR

VAR_INPUT
	SIZE :	UINT;
END_VAR

VAR_OUTPUT
	IS_SORTED :	BOOL;
END_VAR

VAR
	i :	INT;
	i2 :	INT;
	stop :	INT;
END_VAR

(*@KEY@: WORKSHEET
NAME: IS_SORTED
IEC_LANGUAGE: ST
*)
stop :=LIMIT_INT(1,UINT_TO_INT(size),1000);
stop := stop -1;
FOR i := 1 TO stop DO
    i2 := i+1;
	IF pt[i] > pt[i2] THEN
		IS_SORTED := FALSE;
		RETURN;
	END_IF;
END_FOR;

IS_SORTED := TRUE;

(* revision history

hm 	29. mar. 2008 	rev 1.0
	original version

hm	4. apr. 2008	rev 1.1
	added type conversion to avoid warnings under codesys 3.0
*)
(*@KEY@: END_WORKSHEET *)
END_FUNCTION_BLOCK

(* ---- IS_UPPER.ST ---- *)
(*@PROPERTIES_EX@
TYPE: POU
LOCALE: 0
IEC_LANGUAGE: ST
PLC_TYPE: independent
PROC_TYPE: independent
GROUP: STRINGS
*)
(*@KEY@:DESCRIPTION*)
version 1.1	29. mar. 2008
programmer 		kurt
tested by		hugo

IS_UPPER testet ob in einem string keine Kleinbuchstaben vorkommen.
(*@KEY@:END_DESCRIPTION*)
FUNCTION_BLOCK IS_UPPER

(*Group:Default*)

VAR_INPUT
	STR :	STRING;
END_VAR

VAR_OUTPUT
	IS_UPPER :	BOOL;
END_VAR

VAR
	pos :	INT;
	I :	INT;
END_VAR

(*@KEY@: WORKSHEET
NAME: IS_UPPER
IEC_LANGUAGE: ST
*)
I := LEN(str);
FOR pos := 1 TO I DO
	IF NOT ISC_UPPER(INT_TO_BYTE(GET_CHAR(str,pos))) THEN
		IS_UPPER := FALSE;
		RETURN;
	END_IF;
END_FOR;
IS_UPPER := I>0;

(* revision history
hm	29. feb 2008	rev 1.0
	original version

hm	29. mar. 2008	rev 1.1
	changed STRING to STRING(STRING_LENGTH)
*)
(*@KEY@: END_WORKSHEET *)
END_FUNCTION_BLOCK

(* ---- LAMBERT_W.ST ---- *)
(*@PROPERTIES_EX@
TYPE: POU
LOCALE: 0
IEC_LANGUAGE: ST
PLC_TYPE: independent
PROC_TYPE: independent
GROUP: MATHEMATICAL.MATHE
*)
(*@KEY@:DESCRIPTION*)
version 1.1	10. mar. 2009
programmer 	hugo
tested by	oscat

this function calculates the lambert_w function.

(*@KEY@:END_DESCRIPTION*)
FUNCTION_BLOCK LAMBERT_W

(*Group:Default*)

VAR_INPUT
	X :	REAL;
END_VAR

VAR_OUTPUT
	LAMBERT_W :	REAL;
END_VAR

VAR
	w :	REAL;
	i :	INT;
	we :	REAL;
	w1e :	REAL;
	last :	DWORD;
	ewx :	REAL;
END_VAR

(*@KEY@: WORKSHEET
NAME: LAMBERT_W
IEC_LANGUAGE: ST
*)
(* check for valid input and return -1000 if too low *)
IF x < -0.367879441171442 THEN
	LAMBERT_W := -1000.0;
	RETURN;
(* return 0 if x = 0 *)
ELSIF x = 0.0 THEN
	RETURN;
(* first an estimate is calculated *)
ELSIF x <= 500.0 THEN
	w := LN(x + 1.0);
	w := 0.665 * (1.0 + 0.0195 * w) * w + 0.04;
ELSE
	w := LN(x - 4.0) - (1.0 - 1.0/LN(x)) * LN(LN(x));
END_IF;
(* use estimate to calculate exact result *)
FOR i := 0 TO 5 DO
	ewx := EXP(w);
	we := w * ewx - x;
	w1e := (w+1.0) * ewx;
	last := _REAL_TO_DWORD(w) AND DWORD#16#FFFF_FFFC;
	w := w - (we / (w1e - (w+2.0) * we / (2.0 * w + 2.0)));
	IF (_REAL_TO_DWORD(w) AND DWORD#16#FFFF_FFFC) = last THEN EXIT; END_IF;
END_FOR;
LAMBERT_W := w;

(* revision hisdtory
hm	26. oct. 2008	rev 1.0
	original version

hm	10. mar. 2009	rev 1.1
	real constants updated to new systax using dot

*)

(*@KEY@: END_WORKSHEET *)
END_FUNCTION_BLOCK

(* ---- LENGTH.ST ---- *)
(*@PROPERTIES_EX@
TYPE: POU
LOCALE: 0
IEC_LANGUAGE: ST
PLC_TYPE: independent
PROC_TYPE: independent
GROUP: ENGINEERING.CONVERSION
*)
(*@KEY@:DESCRIPTION*)
version 1.1	11. mar. 2009
programmer 	hugo
tested by	oscat

this function converts different length units
any unused input can simply be left open.
different inputs connected at the same time will be added up.
(*@KEY@:END_DESCRIPTION*)
FUNCTION_BLOCK LENGTH

(*Group:Default*)

VAR_INPUT
	M :	REAL;
	P :	REAL;
	IN :	REAL;
	FT :	REAL;
	YD :	REAL;
	MILE :	REAL;
	SM :	REAL;
	FM :	REAL;
END_VAR

VAR_OUTPUT
	YM :	REAL;
	YP :	REAL;
	YIN :	REAL;
	YFT :	REAL;
	YYD :	REAL;
	YMILE :	REAL;
	YSM :	REAL;
	YFM :	REAL;
END_VAR

(*@KEY@: WORKSHEET
NAME: LENGTH
IEC_LANGUAGE: ST
*)
Ym :=	m
		+ p * 0.000376065
		+ in * 0.0254
		+ ft * 0.3048
		+ yd * 0.9144
		+ mile * 1609.344
		+ sm * 1852.0
		+ fm * 1.829;
Yp := Ym * 2659.11478068951;
Yin := Ym * 39.37007874016;
Yft := Ym * 3.28083989501;
Yyd := Ym * 1.09361329834;
Ymile := Ym * 0.00062137119;
Ysm := Ym * 0.00053995680;
Yfm := Ym * 0.54674685621;

(*
Länge Meter m SI-Basiseinheit
Astronomische Einheit* AE 1 AE = 149,597 870 · E9 m
Parsec pc 1 pc = 206265 AE = 30,857 · E15 m
Lichtjahr Lj 1 Lj = 9,460 530 · E15 m = 63240 AE = 0,306 59 pc
Ångström Å 1 Å = E–l0 m
typograph. Punkt p 1 p = 0,376 065 mm • im Druckereigewerbe
inch** in 1 in = 2,54 · E–2 m = 25,4 mm***
foot ft 1 ft = 0,3048 m = 30,48 cm
yard yd 1 yd = 0,9144 m
mile mile 1 mile = 1609,344 m
Internat. Seemeile sm 1 sm = 1852 m
Fathom fm 1 fm = 1,829 m • in der Seeschifffahrt
*)

(* revision history

hm	27. mar. 2007	rev 1.0
	original version

hm	11. mar. 2009	rev 1.1
	improved code

*)

(*@KEY@: END_WORKSHEET *)
END_FUNCTION_BLOCK

(* ---- LINEAR_INT.ST ---- *)
(*@PROPERTIES_EX@
TYPE: POU
LOCALE: 0
IEC_LANGUAGE: ST
PLC_TYPE: independent
PROC_TYPE: independent
GROUP: MATHEMATICAL.FUNCTIONS
*)
(*@KEY@:DESCRIPTION*)
version 1.1	27 dec 2007
programmer 	oscat
tested BY	oscat

LINEAR_INT calculates an output based on a linear interpolation of up to 20 coordinates given in an array
the input coordinates have to start at the lowest array position and must be sorted ba ascending X values.
(*@KEY@:END_DESCRIPTION*)
FUNCTION_BLOCK LINEAR_INT

(*Group:Default*)

VAR_INPUT
	X :	REAL;
	XY :	oscat_XY;
	PTS :	INT;
END_VAR

VAR_OUTPUT
	LINEAR_INT :	REAL;
END_VAR

VAR
	i :	INT;
	i2 :	INT;
END_VAR

(*@KEY@: WORKSHEET
NAME: LINEAR_INT
IEC_LANGUAGE: ST
*)
(*make sure n is bound within the array size *)
pts := MIN(pts,20);

(* calculate the linear segement interpolation *)
i := 2;
(* search for segment and calculate output
	below and above the defined segments we interpolate the last segment *)
WHILE (i < pts) AND (XY[i][0] < X) DO
	i := i + 1;
END_WHILE;

(* Hilfsvariable -> Multiprog erlaubt keine Berechnung innerhalb einer [index] angabe *)
i2 := i-1;

(* calculate the output value on the corresponding segment coordinates *)

LINEAR_INT := ((XY[i][1] - XY[i2][1]) * X - XY[i][1] * XY[i2][0] + XY[i2][1] * XY[i][0]) / (XY[i][0] - XY[i2][0]);

(* revision history
hm	7. oct 2007		rev 1.0
	original version

hm	27 dec 2007		rev 1.1
	changed code for better performance
*)
(*@KEY@: END_WORKSHEET *)
END_FUNCTION_BLOCK

(* ---- LIST_ADD.ST ---- *)
(*@PROPERTIES_EX@
TYPE: POU
LOCALE: 0
IEC_LANGUAGE: ST
PLC_TYPE: independent
PROC_TYPE: independent
GROUP: LIST_PROCESSING
*)
(*@KEY@:DESCRIPTION*)
version 1.0		21. mar. 2011
programmer 	    hugo
tested by		oscat

LIST_ADD hängt ein weiteres element ans ende einer liste.
die liste liegt als string von elementen vor die mit den zeichen SEP am anfang makiert sind.

(*@KEY@:END_DESCRIPTION*)
FUNCTION_BLOCK LIST_ADD

(*Group:Default*)

VAR_INPUT
	SEP :	BYTE;
	INS :	oscat_STRING250;
END_VAR

VAR_IN_OUT
	LIST :	oscat_STRING250;
END_VAR

VAR_OUTPUT
	LIST_ADD :	BOOL;
END_VAR

VAR
	CHR_TO_STRING :	CHR_TO_STRING;
END_VAR

(*@KEY@: WORKSHEET
NAME: LIST_ADD
IEC_LANGUAGE: ST
*)
IF LEN(LIST) + LEN(INS) + 1 <= 250 THEN
  CHR_TO_STRING(C:=SEP);
  LIST := CONCAT(LIST, CHR_TO_STRING.CHR_TO_STRING);
  LIST := CONCAT(LIST, INS);
  LIST_ADD := TRUE;
ELSE
  LIST_ADD := FALSE;
END_IF;

(* revision histroy

hm	21. mar. 2011	rev 2.0
	original release
*)

(*@KEY@: END_WORKSHEET *)
END_FUNCTION_BLOCK

(* ---- LIST_CLEAN.ST ---- *)
(*@PROPERTIES_EX@
TYPE: POU
LOCALE: 0
IEC_LANGUAGE: ST
PLC_TYPE: independent
PROC_TYPE: independent
GROUP: LIST_PROCESSING
*)
(*@KEY@:DESCRIPTION*)
version 2.0	21. mar. 2011
programmer 	hugo
tested by	oscat

LIST_CLEAN bereinigt eine liste von leeren Elementen.
die liste liegt als string von elementen vor die mit den zeichen SEP am anfang markiert sind.

(*@KEY@:END_DESCRIPTION*)
FUNCTION_BLOCK LIST_CLEAN

(*Group:Default*)

VAR_INPUT
	SEP :	BYTE;
END_VAR

VAR_IN_OUT
	LIST :	oscat_STRING250;
END_VAR

VAR_OUTPUT
	LIST_CLEAN :	BOOL;
END_VAR

VAR
	BUF_TO_STRING :	BUF_TO_STRING;
	pt :	oscat_bya_LIST_CLEAN;
	read :	INT;
	write :	INT := 1;
	last :	BYTE;
	c :	BYTE;
	cnt :	INT;
	z :	INT;
END_VAR

(*@KEY@: WORKSHEET
NAME: LIST_CLEAN
IEC_LANGUAGE: ST
*)
last := BYTE#0;
cnt := LEN(LIST);
write := 0;
FOR read := 1 TO cnt DO
	c := INT_TO_BYTE(GET_CHAR(LIST,read));
	IF c <> SEP OR last <> SEP THEN
		write := write + 1;
		pt[write] := c;
	END_IF;
	last := c;
END_FOR;
IF last = SEP THEN write := write - 1; END_IF;

FOR z := 0 TO 1 DO
  BUF_TO_STRING.REQ        := z > 0;
  BUF_TO_STRING.BUF_FORMAT := TRUE;
  BUF_TO_STRING.BUF_OFFS   := DINT#0;
  BUF_TO_STRING.BUF_CNT    := INT_TO_DINT(write);
  BUF_TO_STRING.BUFFER     := pt;
  BUF_TO_STRING.DST        := LIST;
  BUF_TO_STRING();
  pt := BUF_TO_STRING.BUFFER;
  LIST := BUF_TO_STRING.DST;
END_FOR;

LIST_CLEAN := TRUE; (* return TRUE *)

(* revision histroy
hm	28. jun. 2008	rev 1.0
	original release

hm	19. jan. 2011	rev 1.1
	changed string(255) to string(LIST_LENGTH)

hm	21. mar. 2011	rev 2.0
	all elements start with SEP

*)

(*@KEY@: END_WORKSHEET *)
END_FUNCTION_BLOCK

(* ---- LIST_GET.ST ---- *)
(*@PROPERTIES_EX@
TYPE: POU
LOCALE: 0
IEC_LANGUAGE: ST
PLC_TYPE: independent
PROC_TYPE: independent
GROUP: LIST_PROCESSING
*)
(*@KEY@:DESCRIPTION*)
version 2.0	21. mar. 2011
programmer 	hugo
tested by	oscat

LIST_GET liefert das element an der stelle pos einer liste.
die liste liegt als string von elementen vor die mit den zeichen SEP am anfang makiert sind.

(*@KEY@:END_DESCRIPTION*)
FUNCTION_BLOCK LIST_GET

(*Group:Default*)

VAR_INPUT
	SEP :	BYTE;
	POS :	INT;
END_VAR

VAR_IN_OUT
	LIST :	oscat_STRING250;
END_VAR

VAR_OUTPUT
	LIST_GET :	oscat_STRING250;
END_VAR

VAR
	i :	INT;
	i2 :	INT;
	cnt :	INT;
	size :	INT;
END_VAR

(*@KEY@: WORKSHEET
NAME: LIST_GET
IEC_LANGUAGE: ST
*)
cnt := 0;
size := LEN(LIST);

(* search for the n-th occurence of a separation character and store position in i *)
FOR i := 1 TO size DO
    IF cnt = pos THEN EXIT; END_IF;
    IF INT_TO_BYTE(GET_CHAR(LIST,i)) = SEP THEN
        cnt := cnt + 1;
    END_IF;
END_FOR;

FOR i2 := i TO size DO
    IF INT_TO_BYTE(GET_CHAR(LIST,i2)) = SEP THEN EXIT; END_IF;
END_FOR;

IF i2 > i THEN
    LIST_GET := MID(LIST,i2-i,i);
ELSE
    LIST_GET := '';
END_IF;

(* revision histroy
hm	20. jun. 2008	rev 1.0
	original release

hm	19. jan. 2011	rev 1.1
	changed string(255) to strring(LIST_LENGTH)

hm	21. mar. 2011	rev 2.0
	all list elements start with SEP
*)

(*@KEY@: END_WORKSHEET *)
END_FUNCTION_BLOCK

(* ---- LIST_INSERT.ST ---- *)
(*@PROPERTIES_EX@
TYPE: POU
LOCALE: 0
IEC_LANGUAGE: ST
PLC_TYPE: independent
PROC_TYPE: independent
GROUP: LIST_PROCESSING
*)
(*@KEY@:DESCRIPTION*)
version 2.0	21. mar. 2011
programmer 	hugo
tested by	oscat

LIST_INSERT setzt ein element an der stelle pos in eine liste ein.
die liste liegt als string von elementen vor die mit den zeichen SEP am anfang markiert sind.

(*@KEY@:END_DESCRIPTION*)
FUNCTION_BLOCK LIST_INSERT

(*Group:Default*)

VAR_INPUT
	SEP :	BYTE;
	POS :	INT;
	INS :	oscat_STRING250;
END_VAR

VAR_IN_OUT
	LIST :	oscat_STRING250;
END_VAR

VAR_OUTPUT
	LIST_INSERT :	BOOL;
END_VAR

VAR
	cnt :	INT;
	tmp :	oscat_STRING250;
	CHR_TO_STRING :	CHR_TO_STRING;
	size :	INT;
	read :	INT;
	_INSERT :	_INSERT250;
END_VAR

(*@KEY@: WORKSHEET
NAME: LIST_INSERT
IEC_LANGUAGE: ST
*)
CHR_TO_STRING(C:=SEP);
read := 1;
cnt := 1;
size := LEN(LIST);
POS := MAX(POS,1);
LIST_INSERT := FALSE;

WHILE read < 250 DO
	IF cnt = POS THEN
        tmp := CONCAT(CHR_TO_STRING.CHR_TO_STRING, INS);
        _INSERT(IN1:=LIST,IN2:=tmp,P:=read - 1);
        LIST :=_INSERT._INSERT;
		LIST_INSERT := TRUE;
		RETURN;
	END_IF;
	IF read > size THEN
        LIST := CONCAT(LIST,CHR_TO_STRING.CHR_TO_STRING);
        size := size + 1;
    END_IF;
    read := read + 1;
    IF read > size THEN
	    cnt := cnt + 1;
    ELSIF INT_TO_BYTE(GET_CHAR(LIST,read)) = SEP THEN
	    cnt := cnt + 1;
    END_IF;
END_WHILE;

(*@KEY@: END_WORKSHEET *)
END_FUNCTION_BLOCK

(* ---- LIST_LEN.ST ---- *)
(*@PROPERTIES_EX@
TYPE: POU
LOCALE: 0
IEC_LANGUAGE: ST
PLC_TYPE: independent
PROC_TYPE: independent
GROUP: LIST_PROCESSING
*)
(*@KEY@:DESCRIPTION*)
version 2.0	21. mar. 2011
programmer 	hugo
tested by	oscat

LIST_LEN liefert die anzahl der elemente einer liste.
die liste liegt als string von elementen vor die mit den zeichen SEP am anfang markiert sind.

(*@KEY@:END_DESCRIPTION*)
FUNCTION_BLOCK LIST_LEN

(*Group:Default*)

VAR_INPUT
	SEP :	BYTE;
END_VAR

VAR_IN_OUT
	LIST :	oscat_STRING250;
END_VAR

VAR_OUTPUT
	LIST_LEN :	INT;
END_VAR

VAR
	pos :	INT;
	size :	INT;
END_VAR

(*@KEY@: WORKSHEET
NAME: LIST_LEN
IEC_LANGUAGE: ST
*)
size := LEN(LIST);
LIST_LEN := 0;
FOR pos := 1 TO size DO
	IF INT_TO_BYTE(GET_CHAR(LIST,pos)) = SEP THEN LIST_LEN := LIST_LEN + 1; END_IF;
END_FOR;

(* revision histroy
hm	25. jun. 2008	rev 1.0
	original release

hm	16. oct. 2008	rev 1.1
	fixed a problem where list_len would only work up to LIST_LENGTH

hm	19. jan. 2001	rev 1.2
	changed string(255) to string(LIST_LENGTH)

hm	21. mar. 2011	rev 2.0
	all list elements start with SEP

*)

(*@KEY@: END_WORKSHEET *)
END_FUNCTION_BLOCK

(* ---- LIST_NEXT.ST ---- *)
(*@PROPERTIES_EX@
TYPE: POU
LOCALE: 0
IEC_LANGUAGE: ST
PLC_TYPE: independent
PROC_TYPE: independent
GROUP: LIST_PROCESSING
*)
(*@KEY@:DESCRIPTION*)
version 2.0	21. mar. 2011
programmer 	hugo
tested by	oscat

LIST_NEXT retrieves the next element of a list, starting from element 1 after reset or first init.
when the end of the lisat is reached a '' empty string is returned and NUL is set to true.
die liste liegt als string von elementen vor die mit den zeichen SEP am anfang markiert sind.
(*@KEY@:END_DESCRIPTION*)
FUNCTION_BLOCK LIST_NEXT

(*Group:Default*)

VAR_INPUT
	SEP :	BYTE;
	RST :	BOOL;
END_VAR

VAR_IN_OUT
	LIST :	oscat_STRING250;
END_VAR

VAR_OUTPUT
	LEL :	oscat_STRING250;
	NUL :	BOOL;
END_VAR

VAR
	stop :	INT;
	start :	INT;
	pos :	INT := INT#1;
	size :	INT;
END_VAR

(*@KEY@: WORKSHEET
NAME: LIST_NEXT
IEC_LANGUAGE: ST
*)
size := LEN(LIST);
IF rst THEN pos := 1; END_IF;
stop := 0;
start := pos + 1;
stop := pos;
NUL := pos > size;
FOR pos := start TO size DO
	IF INT_TO_BYTE(GET_CHAR(LIST,pos)) = SEP THEN
		EXIT;
	ELSE
		stop := stop + 1;
	END_IF;
END_FOR;
IF stop >= start THEN
	LEL := MID(LIST, stop - start + 1, start);
ELSE
    LEL := '';
END_IF;

(* revision histroy
hm	25. jun. 2008	rev 1.0
	original release

hm	19. jan. 2011	rev 1.1
	changed string(255) to string(LIST_LENGTH)

hm	21. mar. 2011	rev 2.0
	all elements start with SEP

*)

(*@KEY@: END_WORKSHEET *)
END_FUNCTION_BLOCK

(* ---- LIST_RETRIEVE.ST ---- *)
(*@PROPERTIES_EX@
TYPE: POU
LOCALE: 0
IEC_LANGUAGE: ST
PLC_TYPE: independent
PROC_TYPE: independent
GROUP: LIST_PROCESSING
*)
(*@KEY@:DESCRIPTION*)
version 2.0		21. mar. 2011
programmer 	    hugo
tested by		oscat

LIST_RETRIEVE liefert das element an der stelle pos einer liste und löscht das element aus der liste.
die liste liegt als string von elementen vor die mit den zeichen SEP separiert sind.

(*@KEY@:END_DESCRIPTION*)
FUNCTION_BLOCK LIST_RETRIEVE

(*Group:Default*)

VAR_INPUT
	SEP :	BYTE;
	POS :	INT;
END_VAR

VAR_IN_OUT
	LIST :	oscat_STRING250;
END_VAR

VAR_OUTPUT
	LIST_RETRIEVE :	oscat_STRING250;
END_VAR

VAR
	i :	INT;
	cnt :	INT;
	size :	INT;
	z :	INT;
	start :	INT;
	stop :	INT;
END_VAR

(*@KEY@: WORKSHEET
NAME: LIST_RETRIEVE
IEC_LANGUAGE: ST
*)
cnt := 0;
start := 0;
stop := 0;
size := LEN(LIST);
FOR i := 1 TO size DO
	IF INT_TO_BYTE(GET_CHAR(LIST,i)) = SEP THEN
		cnt := cnt + 1;
		IF cnt = POS THEN
			start := i;
			FOR i := start + 1 TO size DO
                IF INT_TO_BYTE(GET_CHAR(LIST,i)) = SEP THEN EXIT; END_IF;
			END_FOR;
			stop := i;
			EXIT;
		END_IF;
	END_IF;
END_FOR;
z := stop - start;
IF z > 1 THEN
	LIST_RETRIEVE := MID(LIST, z - 1, start + 1);
ELSE
	LIST_RETRIEVE := '';
END_IF;
IF z > 0 THEN
	LIST := DELETE(LIST, z, start);
END_IF;

(* revision histroy
hm	28. jun. 2008	rev 1.0
	original release

hm	19. jan. 2011	rev 1.1
	changed string(255) to string(LIST_LENGTH)

hm	21. mar. 2011	rev 2.0
	all elements start with SEP
*)

(*@KEY@: END_WORKSHEET *)
END_FUNCTION_BLOCK

(* ---- LIST_RETRIEVE_LAST.ST ---- *)
(*@PROPERTIES_EX@
TYPE: POU
LOCALE: 0
IEC_LANGUAGE: ST
PLC_TYPE: independent
PROC_TYPE: independent
GROUP: LIST_PROCESSING
*)
(*@KEY@:DESCRIPTION*)
version 2.0		21. mar. 2011
programmer 	    hugo
tested by		oscat

LIST_RETRIEVE liefert das element an der stelle pos einer liste und löscht das element aus der liste.
die liste liegt als string von elementen vor die mit den zeichen SEP separiert sind.

(*@KEY@:END_DESCRIPTION*)
FUNCTION_BLOCK LIST_RETRIEVE_LAST

(*Group:Default*)

VAR_INPUT
	SEP :	BYTE;
END_VAR

VAR_IN_OUT
	LIST :	oscat_STRING250;
END_VAR

VAR_OUTPUT
	LIST_RETRIEVE_LAST :	oscat_STRING250;
END_VAR

VAR
	i :	INT;
	size :	INT;
END_VAR

(*@KEY@: WORKSHEET
NAME: LIST_RETRIEVE_LAST
IEC_LANGUAGE: ST
*)
size := LEN(LIST);
i := size;
WHILE i > 0 DO
	IF INT_TO_BYTE(GET_CHAR(LIST,i)) = SEP THEN
        LIST_RETRIEVE_LAST := RIGHT(LIST, size - i);
        LIST := LEFT(LIST, i - 1);
		RETURN;
    ELSE
        i := i - 1;
    END_IF;
END_WHILE;
LIST_RETRIEVE_LAST := '';
LIST := '';

(* revision histroy
hm	21. mar. 2011	rev 2.0
	new module
*)

(*@KEY@: END_WORKSHEET *)
END_FUNCTION_BLOCK

(* ---- LOWERCASE.ST ---- *)
(*@PROPERTIES_EX@
TYPE: POU
LOCALE: 0
IEC_LANGUAGE: ST
PLC_TYPE: independent
PROC_TYPE: independent
GROUP: STRINGS
*)
(*@KEY@:DESCRIPTION*)
version 1.3	29. mar. 2008
programmer 	hugo
tested by		tobias

lowercase returns str while all letters A..Z and Ä.Ö,Ü are converted to lowercase.
(*@KEY@:END_DESCRIPTION*)
FUNCTION_BLOCK LOWERCASE

(*Group:Default*)

VAR_INPUT
	STR :	STRING;
END_VAR

VAR_OUTPUT
	LOWERCASE :	STRING;
END_VAR

VAR
	char :	BYTE;
	char2 :	BYTE;
	pos :	INT;
	l :	INT;
	str_temp :	STRING;
END_VAR

(*@KEY@: WORKSHEET
NAME: LOWERCASE
IEC_LANGUAGE: ST
*)
LOWERCASE := str;
l := LEN(str);
FOR pos := 1 TO l DO
    char := INT_TO_BYTE(GET_CHAR(str,pos));
	char2 := TO_LOWER(char);
    IF char <> char2 THEN
    	str_temp := LOWERCASE;
      	LOWERCASE := REPLACE(str_temp,BYTE_TO_STRING(char2,'%c'),1,pos);
	END_IF;
END_FOR;

(* revision histroy
hm	6. oct. 2006	rev 1.0
	original release

hm	4. feb. 2008	rev 1.1
	improved performance
	added Ä.Ö,Ü

hm	6. mar. 2008	rev 1.2
	added support for exteded Ascii

hm	29. mar. 2008	rev 1.3
	changed STRING to STRING(STRING_LENGTH)
*)
(*@KEY@: END_WORKSHEET *)
END_FUNCTION_BLOCK

(* ---- LTCH.ST ---- *)
(*@PROPERTIES_EX@
TYPE: POU
LOCALE: 0
IEC_LANGUAGE: ST
PLC_TYPE: independent
PROC_TYPE: independent
GROUP: LOGIC.FF_PULSE_TRIGGERED
*)
(*@KEY@:DESCRIPTION*)
version 1.2	30. oct. 2008
programmer 	hugo
tested by	oscat

Transparent Latch with asynchronous reset
(*@KEY@:END_DESCRIPTION*)
FUNCTION_BLOCK LTCH

(*Group:Default*)

VAR_INPUT
	D :	BOOL;
	L :	BOOL;
	RST :	BOOL;
END_VAR

VAR_OUTPUT
	Q :	BOOL;
END_VAR

(*@KEY@: WORKSHEET
NAME: LTCH
IEC_LANGUAGE: ST
*)
(* as long as L is true, the latch is transparent and and change of D is transferred to Q *)
(* of course only when there is no asynchronous reset *)
IF rst THEN				(* if asynchronous reset then Q=0 *)
	Q := FALSE;
ELSIF L THEN			(* latch is transparent *)
	Q := D;
END_IF;

(* revision history
hm	4. aug 2006		rev 1.0
	original version

hm	27. dec 2007	rev 1.1
	changed code for better performance

hm	30. oct. 2008	rev 1.2
	deleted unnecessary init with 0

*)
(*@KEY@: END_WORKSHEET *)
END_FUNCTION_BLOCK

(* ---- LTCH_4.ST ---- *)
(*@PROPERTIES_EX@
TYPE: POU
LOCALE: 0
IEC_LANGUAGE: ST
PLC_TYPE: independent
PROC_TYPE: independent
GROUP: LOGIC.FF_PULSE_TRIGGERED
*)
(*@KEY@:DESCRIPTION*)
version 1.3	14. mar. 2009
programmer 	hugo
tested by	oscat

Quad Transparent Latch with asynchronous reset
(*@KEY@:END_DESCRIPTION*)
FUNCTION_BLOCK LTCH_4

(*Group:Default*)

VAR_INPUT
	D0 :	BOOL;
	D1 :	BOOL;
	D2 :	BOOL;
	D3 :	BOOL;
	L :	BOOL;
	RST :	BOOL;
END_VAR

VAR_OUTPUT
	Q0 :	BOOL;
	Q1 :	BOOL;
	Q2 :	BOOL;
	Q3 :	BOOL;
END_VAR

(*@KEY@: WORKSHEET
NAME: LTCH_4
IEC_LANGUAGE: ST
*)
(* as long as L is true, the latch is transparent and and change of D is transferred to Q *)
(* of course only when there is no asynchronous reset *)
IF rst THEN			(* if asynchronous reset then Q=0 *)
	Q0 := FALSE;
	Q1 := FALSE;
	Q2 := FALSE;
	Q3 := FALSE;
ELSIF L THEN			(* latch is transparent *)
	Q0 := D0;
	Q1 := D1;
	Q2 := D2;
	Q3 := D3;
END_IF;

(* revision history
hm	4. aug 2006	rev 1.0
	original version

hm	27. dec 2007	rev 1.1
	changed code for better performance

hm	30. oct. 2008	rev 1.2
	deleted unnecessary init with 0

hm	14. mar. 2009	rev 1.3
	removed double assignments

*)
(*@KEY@: END_WORKSHEET *)
END_FUNCTION_BLOCK

(* ---- M_D.ST ---- *)
(*@PROPERTIES_EX@
TYPE: POU
LOCALE: 0
IEC_LANGUAGE: ST
PLC_TYPE: independent
PROC_TYPE: independent
GROUP: ENGINEERING.MEASUREMENTS
*)
(*@KEY@:DESCRIPTION*)
version 1.2	27. feb. 2009
programmer 	hugo
tested BY	oscat

m_d measures the time between a rising edge on start to a rising edge on stop and returs the last measured value on the output PT.
a second output ET is starting from 0 at the rising edge of start and is counting up until the rising edge of stop occurs.
the asynchronous input rst can reset the outputs at any time.
tmax defines a timeout wich is the maximum measurable time between start and stop, if this time is exceeded the outputs will stay at 0.
(*@KEY@:END_DESCRIPTION*)
FUNCTION_BLOCK M_D

(*Group:Default*)

VAR_INPUT
	START :	BOOL;
	STOP :	BOOL;
	TMAX :	TIME := t#10d;
	RST :	BOOL;
END_VAR

VAR_OUTPUT
	PT :	TIME;
	ET :	TIME;
	RUN :	BOOL;
END_VAR

VAR
	edge :	BOOL;
	T0 :	TIME;
	tx :	TIME;
	startup :	BOOL;
	T_PLC_MS :	T_PLC_MS;
END_VAR

(*@KEY@: WORKSHEET
NAME: M_D
IEC_LANGUAGE: ST
*)
(* check for rst input *)
IF rst OR et >= tmax THEN
	pt := t#0ms;
	et := t#0ms;
	startup := FALSE;
	run := FALSE;
END_IF;

(* avoid timers to start when input is true at startup *)
IF NOT startup THEN
	edge := start;
	startup := TRUE;
END_IF;

(* read system timer *)
T_PLC_MS();
tx:= UDINT_TO_TIME(T_PLC_MS.T_PLC_MS);

(* detect rising edge on start *)
IF start AND NOT edge AND NOT stop THEN
	t0 := tx;
	run := TRUE;
	pt := t#0s;
ELSIF stop AND run THEN
	pt := et;
	run := FALSE;
END_IF;
edge := start;
IF run THEN et := tx - t0; END_IF;

(* revision history
hm		2.5.2007	rev 1.0
	original version

hm		16.9.2007	rev 1.1
	changes time() to T_plc_ms() for compatibility reasons

hm	27. feb 2009	rev 1.2
	deleted unnecessary init with 0
*)
(*@KEY@: END_WORKSHEET *)
END_FUNCTION_BLOCK

(* ---- M_T.ST ---- *)
(*@PROPERTIES_EX@
TYPE: POU
LOCALE: 0
IEC_LANGUAGE: ST
PLC_TYPE: independent
PROC_TYPE: independent
GROUP: ENGINEERING.MEASUREMENTS
*)
(*@KEY@:DESCRIPTION*)
version 1.4	10. mar. 2009
programmer 	hugo
tested BY	oscat

m_t measures the with of a high pulse and returs the last measured pulse width on output PT.
a second output ET is starting from 0 at the rising edge and counting up until the falling edge occurs and resetts et to 0.
the asynchrtonous input rst can reset the outputs at any time.
tmax defines a maximum measurable time, if this value is exceeded the outputs will be reset to 0.

(*@KEY@:END_DESCRIPTION*)
FUNCTION_BLOCK M_T

(*Group:Default*)

VAR_INPUT
	IN :	BOOL;
	TMAX :	TIME := t#10d;
	RST :	BOOL;
END_VAR

VAR_OUTPUT
	PT :	TIME;
	ET :	TIME;
END_VAR

VAR
	edge :	BOOL;
	start :	TIME;
	tx :	TIME;
	T_PLC_MS :	T_PLC_MS;
END_VAR

(*@KEY@: WORKSHEET
NAME: M_T
IEC_LANGUAGE: ST
*)
(* read system timer *)
T_PLC_MS();
tx:= UDINT_TO_TIME(T_PLC_MS.T_PLC_MS);

IF RST OR ET >= TMAX THEN
	PT := t#0s;
	ET := PT;
ELSIF IN THEN
	IF NOT edge THEN start := tx; END_IF;
	ET := tx - start;
ELSE
	PT := ET;
END_IF;
edge := IN;

(* revision history
hm	4. aug. 2006	rev 1.0
	original version

hm	2. may. 2007	rev 1.1
	added init variable to avoid unreasonable measurement if falling edge occurs first.
	added et (elapsed time) output to count from 0 at rising edge until a falling edge resets et to 0.
	added reset input.

hm	16. sep. 2007	rev 1.2
	changes time() to T_plc_ms() for compatibility reasons

hm	17. dec. 2008	rev 1.3
	code optimized

hm	10. mar. 2009	rev 1.4
	removed nested comments

*)
(*@KEY@: END_WORKSHEET *)
END_FUNCTION_BLOCK

(* ---- M_TX.ST ---- *)
(*@PROPERTIES_EX@
TYPE: POU
LOCALE: 0
IEC_LANGUAGE: ST
PLC_TYPE: independent
PROC_TYPE: independent
GROUP: ENGINEERING.MEASUREMENTS
*)
(*@KEY@:DESCRIPTION*)
version 1.4	11. mar. 2009
programmer 	oscat
tested BY	oscat

this measures the timing of a signal
TH is the high pulse width
TL is the low pulse width
DC is the duty cycle
F is the frequency
ET will start at 0 with a rising edge and count up till the next rising edge starts from 0 again.
the acuracy depends on the cycle time of the sps and is limited to 1ms resolution.
an asynchronous reset can reset all outputs to 0 at any time.
the input tmax can configure a timeout for ET where the function block will outomatically reset itself.
tmx is predefined to 10 days.
(*@KEY@:END_DESCRIPTION*)
FUNCTION_BLOCK M_TX

(*Group:Default*)

VAR_INPUT
	IN :	BOOL;
	TMAX :	TIME := t#10d;
	RST :	BOOL;
END_VAR

VAR_OUTPUT
	TH :	TIME;
	TL :	TIME;
	DC :	REAL;
	F :	REAL;
	ET :	TIME;
END_VAR

VAR
	edge :	BOOL;
	start :	TIME;
	stop :	TIME;
	tx :	TIME;
	rise :	BOOL;
	fall :	BOOL;
	startup :	BOOL;
	T_PLC_MS :	T_PLC_MS;
END_VAR

(*@KEY@: WORKSHEET
NAME: M_TX
IEC_LANGUAGE: ST
*)
(* check FOR rst input *)
IF rst OR (et >= tmax) THEN
	rise := FALSE;
	fall := FALSE;
	startup := FALSE;
	th := t#0ms;
	tl := t#0ms;
	DC := 0.0;
	F := 0.0;
	ET := t#0s;
END_IF;

(* avoid timers to start when input is true at startup *)
IF NOT startup THEN
	edge := in;
	startup := TRUE;
END_IF;

(* read system timer *)
T_PLC_MS();
tx:= UDINT_TO_TIME(T_PLC_MS.T_PLC_MS);

(* edge trigger rising and falling edge *)
IF in XOR edge THEN
	edge := in;
	(* rising edge starts measurement *)
	IF in THEN
		start := Tx;
		rise := TRUE;
		IF fall THEN tl := start - stop; END_IF;
		IF th > t#0ms AND tl > t#0ms THEN
			dc := TIME_TO_REAL(th) / TIME_TO_REAL(th+tl);
			f := 1000.0 / TIME_TO_REAL(th + tl);
		END_IF;
	(* falling edge starts second cycle measurement *)
	ELSE
		stop := Tx;
		fall := TRUE;
		IF rise THEN th := stop - start; END_IF;
		IF th > t#0ms AND tl > t#0ms THEN
			dc := TIME_TO_REAL(th) /  TIME_TO_REAL(th+tl);
			f := 1000.0 / TIME_TO_REAL(th + tl);
		END_IF;
	END_IF;
END_IF;
IF rise THEN et := tx - start; END_IF;

(* revision history
hm	4. aug. 2006	rev 1.0
	original version

hm	2. mai. 2007	rev 1.1
	made sure that no undefined values would be measured at startup conditions
	added output et
	added rst input
	added tmax input

hm	16. sep. 2007	rev 1.2
	changes time() to T_plc_ms() for compatibility reasons

hm	27. feb. 2009	rev 1.3
	deleted unnecessary init with 0

hm	11. mar. 2009	rev 1.4
	changed real constants to use dot syntax

*)

(* check FOR rst input *)
IF rst OR (et >= tmax) THEN
	rise := FALSE;
	fall := FALSE;
	startup := FALSE;
	th := t#0ms;
	tl := t#0ms;
	DC := 0.0;
	F := 0.0;
	ET := t#0s;
END_IF;

(* avoid timers to start when input is true at startup *)
IF NOT startup THEN
	edge := in;
	startup := TRUE;
END_IF;

(* read system timer *)
T_PLC_MS();
tx:= UDINT_TO_TIME(T_PLC_MS.T_PLC_MS);

(* edge trigger rising and falling edge *)
IF in XOR edge THEN
	edge := in;
	(* rising edge starts measurement *)
	IF in THEN
		start := Tx;
		rise := TRUE;
		IF fall THEN tl := start - stop; END_IF;
		IF th > t#0ms AND tl > t#0ms THEN
			dc := TIME_TO_REAL(th) / TIME_TO_REAL(th+tl);
			f := 1000.0 / TIME_TO_REAL(th + tl);
		END_IF;
	(* falling edge starts second cycle measurement *)
	ELSE
		stop := Tx;
		fall := TRUE;
		IF rise THEN th := stop - start; END_IF;
		IF th > t#0ms AND tl > t#0ms THEN
			dc := TIME_TO_REAL(th) /  TIME_TO_REAL(th+tl);
			f := 1000.0 / TIME_TO_REAL(th + tl);
		END_IF;
	END_IF;
END_IF;
IF rise THEN et := tx - start; END_IF;

(* revision history
hm	4. aug. 2006	rev 1.0
	original version

hm	2. mai. 2007	rev 1.1
	made sure that no undefined values would be measured at startup conditions
	added output et
	added rst input
	added tmax input

hm	16. sep. 2007	rev 1.2
	changes time() to T_plc_ms() for compatibility reasons

hm	27. feb. 2009	rev 1.3
	deleted unnecessary init with 0

*)
(*@KEY@: END_WORKSHEET *)
END_FUNCTION_BLOCK

(* ---- MANUAL_1.ST ---- *)
(*@PROPERTIES_EX@
TYPE: POU
LOCALE: 0
IEC_LANGUAGE: ST
PLC_TYPE: independent
PROC_TYPE: independent
GROUP: ENGINEERING.AUTOMATION
*)
(*@KEY@:DESCRIPTION*)
version 1.2	14. mar. 2009
programmer 	hugo
tested by	oscat

MANUAL_1 is a manual override for digital signals.
When MAN = FALSE, the output follows IN and when MAN = TRUE the Output follows M_I.

(*@KEY@:END_DESCRIPTION*)
FUNCTION_BLOCK MANUAL_1

(*Group:Default*)

VAR_INPUT
	IN :	BOOL;
	MAN :	BOOL;
	M_I :	BOOL;
	SET :	BOOL;
	RST :	BOOL;
END_VAR

VAR_OUTPUT
	Q :	BOOL;
	STATUS :	BYTE;
END_VAR

VAR
	S_edge :	BOOL;
	r_edge :	BOOL;
	edge :	BOOL;
END_VAR

(*@KEY@: WORKSHEET
NAME: MANUAL_1
IEC_LANGUAGE: ST
*)
IF NOT man THEN
	Q := IN;
	STATUS := BYTE#100;
	edge := FALSE;
ELSIF NOT s_edge AND set THEN
	Q := TRUE;
	edge := TRUE;
	status := BYTE#101;
ELSIF NOT r_edge AND rst THEN
	Q := FALSE;
	edge := TRUE;
	status := BYTE#102;
ELSIF NOT edge THEN
	Q := M_I;
	status := BYTE#103;
END_IF;

(* remember levels of manual signals *)
s_edge := SET;
r_edge := RST;

(* revision history
hm	17. jun 2008	rev 1.0
	original version

hm	17. oct 2008	rev 1.1
	deleted unnecessary variable m_edge

hm	14. mar. 2009	rev 1.2
	replaced double assignments

*)
(*@KEY@: END_WORKSHEET *)
END_FUNCTION_BLOCK

(* ---- MANUAL_2.ST ---- *)
(*@PROPERTIES_EX@
TYPE: POU
LOCALE: 0
IEC_LANGUAGE: ST
PLC_TYPE: independent
PROC_TYPE: independent
GROUP: ENGINEERING.AUTOMATION
*)
(*@KEY@:DESCRIPTION*)
version 1.0	22. sep. 2008
programmer 	hugo
tested by	oscat

MANUAL_2 is a manual override for boolean signals.
it has static force high and low as well as a manual input.
(*@KEY@:END_DESCRIPTION*)
FUNCTION_BLOCK MANUAL_2

(*Group:Default*)

VAR_INPUT
	IN :	BOOL;
	ENA :	BOOL;
	ON :	BOOL;
	OFF :	BOOL;
	MAN :	BOOL;
END_VAR

VAR_OUTPUT
	Q :	BOOL;
	STATUS :	BYTE;
END_VAR

(*@KEY@: WORKSHEET
NAME: MANUAL_2
IEC_LANGUAGE: ST
*)
IF ena THEN
	IF NOT ON AND NOT OFF THEN
		Q := IN;
		STATUS := BYTE#100;
	ELSIF on AND NOT off THEN
		Q := TRUE;
		STATUS := BYTE#101;
	ELSIF NOT on AND off THEN
		q := FALSE;
		STATUS := BYTE#102;
	ELSE
		Q := MAN;
		STATUS := BYTE#103;
	END_IF;
ELSE
	Q := FALSE;
	STATUS := BYTE#104;
END_IF;

(* revision history
hm	22. sep. 2008		rev 1.0
	original version

*)
(*@KEY@: END_WORKSHEET *)
END_FUNCTION_BLOCK

(* ---- MANUAL_4.ST ---- *)
(*@PROPERTIES_EX@
TYPE: POU
LOCALE: 0
IEC_LANGUAGE: ST
PLC_TYPE: independent
PROC_TYPE: independent
GROUP: ENGINEERING.AUTOMATION
*)
(*@KEY@:DESCRIPTION*)
version 1.0	17. jun 2008
programmer 	hugo
tested by	oscat

MANUAL_4 is a manual override for digital signals.
When MAN = FALSE, the output follows IN and when MAN = TRUE the Output follows M_I.
(*@KEY@:END_DESCRIPTION*)
FUNCTION_BLOCK MANUAL_4

(*Group:Default*)

VAR_INPUT
	I0 :	BOOL;
	I1 :	BOOL;
	I2 :	BOOL;
	I3 :	BOOL;
	MAN :	BOOL;
	STP :	BOOL;
	M0 :	BOOL;
	M1 :	BOOL;
	M2 :	BOOL;
	M3 :	BOOL;
END_VAR

VAR_OUTPUT
	Q0 :	BOOL;
	Q1 :	BOOL;
	Q2 :	BOOL;
	Q3 :	BOOL;
	STATUS :	BYTE;
END_VAR

VAR
	edge :	BOOL;
	pos :	INT;
	tog :	BOOL;
END_VAR

(*@KEY@: WORKSHEET
NAME: MANUAL_4
IEC_LANGUAGE: ST
*)
IF man THEN
	IF NOT TOG THEN
		Q0 := M0;
		Q1 := M1;
		Q2 := M2;
		Q3 := M3;
		STATUS := BYTE#101;
	END_IF;
	IF STP AND NOT edge THEN
		tog := TRUE;
		CASE pos OF
			0:	Q0 := TRUE;
				Q1 := FALSE;
				Q2 := FALSE;
				Q3 := FALSE;
				STATUS := BYTE#110;
			1:	Q0 := FALSE;
				Q1 := TRUE;
				Q2 := FALSE;
				Q3 := FALSE;
				STATUS := BYTE#111;
			2:	Q0 := FALSE;
				Q1 := FALSE;
				Q2 := TRUE;
				Q3 := FALSE;
				STATUS := BYTE#112;
			3:	Q0 := FALSE;
				Q1 := FALSE;
				Q2 := FALSE;
				Q3 := TRUE;
				STATUS := BYTE#113;
		END_CASE;
		pos := INC(pos,1,3);
	END_IF;
ELSE
	Q0 := I0;
	Q1 := I1;
	Q2 := I2;
	Q3 := I3;
	STATUS := BYTE#100;
	tog := FALSE;
	pos := 0;
END_IF;

(* remember status of stp *)
edge := STP;

(* revision history
hm	17. jun 2008		rev 1.0
	original version

*)
(*@KEY@: END_WORKSHEET *)
END_FUNCTION_BLOCK
